# B&R Automation Studio project RS15_RX_30005_r00 (part 5)

#### A5_AutomatCyclic.st - Cyclic code
```iecst
 (********************************************************************
 * COPYRIGHT -- Microsoft
 ********************************************************************
 * Program: A5_Automat
 * File: A5_AutomatCyclic.st
 * Author: pkiel
 * Created: July 13, 2011
 ********************************************************************
 * Implementation of program A5_Automat
 ********************************************************************)

PROGRAM _CYCLIC

  // Synchro ratio Master/Slave
     // Master = Virtuel
     gA[5].rRSynNum := gRecipeActive.Repeat ;
     gA[5].rRSynDen := g_rSizeEntryPullRol_mm / 25.4 ;

  // Signal synchro Holding axis
  MC_BR_AutControl_0.Signal2 := gA[3].Ind_bSynchroOK                       AND
                                (MC_BR_AutControl_0.ActualStateIndex = 10) ;
  MC_BR_AutControl_0.Signal3 := NOT(gA[3].Ind_bSynchroOK) ;

  // Gear ratio assignement
  IF gReg[5].Enable THEN
    rGearValue := gReg[5].SP_Repeat * gA[5].UnitsPerInch ;
  ELSE
    rGearValue := gA5_GearValue ;
  END_IF

(**** STRAIGHT GEARED CAM AUTOMAT WITH GEARING UPDATE AND NO ABSOLUTE PHASE SYNCHRONIZATION ***)

(* Set Up Master Position Parameter ID *)
  //Synch_Request := gA[5].Cmd_SynchronizedMotion ;
  Synch_Request := gA[5].Cmd_SynchronizedMotion AND NOT(MC_BR_AutControl_0.Stop) ;  // D.M. 26/01/2012 RS26 Pyrollpack_14661 added because after guard fault it happened that Stop=1 and Synch_Request=1 => MC_BR_AutControl_0 makes fault 29256
	IF (Synch_Request AND NOT ParID_Ready) THEN
		MC_BR_InitMasterParIDTransfer_0.Master:=gA[9].Ident;
	    MC_BR_InitMasterParIDTransfer_0.Slave:=gA[5].Ident;
	    MC_BR_InitMasterParIDTransfer_0.MasterParID:=412;
	    MC_BR_InitMasterParIDTransfer_0.SlaveChannel:=0;
	    MC_BR_InitMasterParIDTransfer_0.Execute:=TRUE;
	    IF (MC_BR_InitMasterParIDTransfer_0.Done) THEN
	      MasterParID:=MC_BR_InitMasterParIDTransfer_0.ReceiveParID;
	      MC_BR_InitMasterParIDTransfer_0.Execute:=FALSE;
	      ParID_Ready:=1;
	    ELSIF (MC_BR_InitMasterParIDTransfer_0.Error) THEN
	    (*Store ErrorID in a variable,
	      ErrorID is reset on falling edge of 'Execute'*)
	      ErrorID:=MC_BR_InitMasterParIDTransfer_0.ErrorID;
	      ParID_Ready:=0;
	      MC_BR_InitMasterParIDTransfer_0.Execute:=FALSE;
	    END_IF
	END_IF
	MC_BR_InitMasterParIDTransfer_0();

(**** Initialize Automat Parameters Upon Automat Start Request ****)

	IF (EDGEPOS(ParID_Ready))THEN
		(*general automat parameter*)
			(*AutData.Master				:= gA[1].Ident;*)
			AutData.MasterParID			:= MasterParID;
			AutData.StartPosition		:= 0;
			AutData.StartInterval		:= gA[9].AxisPeriod;
			AutData.MaxMasterVelocity	:= gr_rMachMaxSpeed_BPM ;

		(*Automat STATE 0 Basis State*)
			AutData.State[0].Event[0].Type		  := ncST_END;
			AutData.State[0].Event[0].Attribute	:= ncAT_ONCE;
			//AutData.State[0].Event[0].NextState	:= 1;
      AutData.State[0].Event[0].NextState  := 10;

    //Waiting synchro Holding axis
      AutData.State[10].CamProfileIndex := 16#FFFF;
      AutData.State[10].MasterFactor    := REAL_TO_UDINT(gA[9].AxisPeriod);
      AutData.State[10].SlaveFactor     := 0;
      AutData.State[10].CompMode        := ncOFF;

      AutData.State[10].Event[0].Type      := ncSIGNAL3 ;
      AutData.State[10].Event[0].Attribute := ncAT_ONCE ;
      AutData.State[10].Event[0].NextState := 0;

      AutData.State[10].Event[0].Type      := ncSIGNAL2 ;
      AutData.State[10].Event[0].Attribute := ncAT_ONCE ;
      AutData.State[10].Event[0].NextState := 1;

		(*Automat STATE 1 Master/Slave Run*)
			AutData.State[1].CamProfileIndex := 16#FFFF;
			AutData.State[1].MasterFactor		 := REAL_TO_UDINT(gA[9].AxisPeriod);
			AutData.State[1].SlaveFactor		 := REAL_TO_UDINT(rGearValue);
			AutData.State[1].CompMode			   := ncOFF;

			AutData.State[1].Event[0].Type		:= ncST_END;
			AutData.State[1].Event[0].Attribute	:= ncST_END;
			AutData.State[1].Event[0].NextState	:= 1;

			AutData.State[1].Event[1].Type		:= ncST_END+ncNEGATIVE;
			AutData.State[1].Event[1].Attribute	:= ncST_END;
			AutData.State[1].Event[1].NextState	:= 1;

      AutData.State[1].Event[2].Type    := ncSIGNAL1;
      AutData.State[1].Event[2].Attribute  := ncAT_ONCE;
      AutData.State[1].Event[2].NextState  := 1;

      AutData.State[1].Event[3].Type    := ncSIGNAL3;
      AutData.State[1].Event[3].Attribute  := ncAT_ONCE;
      AutData.State[1].Event[3].NextState  := 0;

			MC_BR_AutControl_0.Enable 		:= 1;
			MC_BR_AutControl_0.AdrAutData 	:= ADR(AutData);
			MC_BR_AutControl_0.InitAutData 	:= 1;
	END_IF

		(* wait for initialization done *)
			IF ((MC_BR_AutControl_0.AutDataInitialized = 1)AND(Synch_Request)) THEN
				MC_BR_AutControl_0.InitAutData 	:= 0;
        uiMC_BR_AutControl_0_MemoErrorID := 0 ;
				AutomatStart := 1;
			END_IF
		(* check if error occured *)
			IF (MC_BR_AutControl_0.ErrorID <> 0) THEN
				MC_BR_AutControl_0.Enable := 0;
        uiMC_BR_AutControl_0_MemoErrorID := MC_BR_AutControl_0.ErrorID ;
			END_IF

(******************** ENABLE CAM-AUTOMAT **********************)
	IF (AutomatStart) THEN
			MC_BR_AutControl_0.Start := 1;
			AutomatStart := 0;
	END_IF

	IF (NOT Synch_Request) THEN
			MC_BR_AutControl_0.Stop := 1;
			MC_BR_AutControl_0.Start := 0;
			ParID_Ready := 0;
      IF (MC_BR_AutControl_0.Running=0) AND
         MC_BR_AutControl_0.Stop        THEN
        MC_BR_AutControl_0.Enable := 0;
        MC_BR_AutControl_0.Stop := 0;
      END_IF
   //*************************************************
   // D.M. 26/01/2012 RS26 Pyrollpack_14661 added because after guard fault it happened that Stop=1 and MC_BR_AutControl_0.Enable => not possible to finish MC_BR_AutControl_0 => program locked
      IF MC_BR_AutControl_0.Stop        AND
         NOT(MC_BR_AutControl_0.Enable) THEN
        MC_BR_AutControl_0.Enable := 1 ;
      END_IF
   //*************************************************
	END_IF
	gA[5].Ind_AutomatEnabled:=MC_BR_AutControl_0.Enable;
	gA[5].Ind_CurrentAutomatState:=MC_BR_AutControl_0.ActualStateIndex;
  gA[5].Ind_bSynchroOK := (MC_BR_AutControl_0.ActualStateIndex = 1) AND gA[5].Ind_SynchronizedMotion ;

(********************** MC_AUTCONTROL *************************)
	MC_BR_AutControl_0.Slave:= gA[5].Ident;
	MC_BR_AutControl_0();

(******************** UPDATE CAM-AUTOMAT STATE 1 **********************)
	MC_BR_InitAutState_0.MasterParID := MasterParID;
	MC_BR_InitAutState_0.Slave := gA[5].Ident;
	MC_BR_InitAutState_0.StateIndex := 1;
	MC_BR_InitAutState_0.CamProfileIndex := 16#FFFF;
	MC_BR_InitAutState_0.MasterFactor := REAL_TO_UDINT(gA[9].AxisPeriod);
	MC_BR_InitAutState_0.SlaveFactor := REAL_TO_DINT(rGearValue);
	MC_BR_InitAutState_0.CompMode := ncOFF;
	MC_BR_InitAutState_0.Execute := gA[5].Cmd_SynchronizedMotionUpdate;
	MC_BR_InitAutState_0();

  IF gA[5].Cmd_SynchronizedMotionUpdate THEN
    iTest_[2] := iTest_[2] + 1 ;
  END_IF

	IF (MC_BR_InitAutState_0.Done) THEN
		gA[5].Cmd_SynchronizedMotionUpdate:=0;
		MC_BR_AutControl_0.Signal1:=1;
    iTest_[0] := iTest_[0] + 1 ;
	ELSE
		MC_BR_AutControl_0.Signal1:=0;
	END_IF

  IF (MC_BR_InitAutState_0.Error) THEN
    gA[5].Cmd_SynchronizedMotionUpdate:=0;
    MC_BR_InitAutState_0.Execute := 0;
    iTest_[1] := iTest_[1] + 1 ;
  END_IF

END_PROGRAM
```

#### A5_Automat.var - Local variables
```iecst
(********************************************************************
 * COPYRIGHT -- Microsoft
 ********************************************************************
 * Program: A5_Automat
 * File: A5_Automat.var
 * Author: pkiel
 * Created: July 13, 2011
 ********************************************************************
 * Local variables of program A5_Automat
 ********************************************************************)
VAR
	AutData : MC_AUTDATA_TYP;
	AutomatStart : BOOL;
	ErrorID : UINT;
	MasterParID : UINT;
	MC_BR_AutControl_0 : MC_BR_AutControl;
  uiMC_BR_AutControl_0_MemoErrorID : UINT := 0 ;
	MC_BR_InitAutState_0 : MC_BR_InitAutState;
	MC_BR_InitMasterParIDTransfer_0 : MC_BR_InitMasterParIDTransfer;
	ParID_Ready : BOOL;
	Synch_Request : BOOL;

  iTest_ : ARRAY[0..9] OF INT ;
  rGearValue : REAL ;
END_VAR
```

### Program Logical/BagMachine_Section/EntryPull/Axis5/A5_Draw (IEC) - Axis Draw Calculations

#### A5_Draw.var - Local variables
```iecst
(********************************************************************
 * COPYRIGHT -- Microsoft
 ********************************************************************
 * Program: A5_Draw
 * File: A5_Draw.var
 * Author: pkiel
 * Created: July 13, 2011
 ********************************************************************
 * Local variables of program A5_Draw
 ********************************************************************)
VAR
	Draw_Old : REAL;
	First : BOOL;
  iLockEntryWebDraw : INT ;
  iBackColor : INT ;

  rEntry_Draw_Nul     : REAL := 0.0;
  rEntry_Draw_SP      : REAL := 0.0;
  HMI_rEntry_Draw_Set : REAL ;
END_VAR
```

### Program Logical/BagMachine_Section/EntryPull/Registration/A5_Reg1 (IEC) - Entry Pull Roll Registration

#### A5_Reg1Init.st
```iecst
(********************************************************************
 * COPYRIGHT -- Microsoft
 ********************************************************************
 * Program: A5_Reg1
 * File: A5_Reg1Init.st
 * Author: pkiel
 * Created: July 19, 2011
 ********************************************************************
 * Implementation of program A5_Reg1
 ********************************************************************)

PROGRAM _INIT

(*Set MC_BR_TouchProbe_0 Block to Capture Virtual Master Commanded Position (Par ID 412) *)
	TriggerRef_0.ProbeParID:=412;

(*Set MC_BR_TouchProbe_0 Block to Hardwired Trigger #1*)
	TriggerRef_0.EventSourceParID:=ACP10PAR_STAT_TRIGGER1;

(*Set MC_BR_TouchProbe_0 Block Trigger For Positive Edge *)
	TriggerRef_0.Edge:=0;

(*Set MC_BR_TouchProbe_1 Block to Capture Encoder #1 Actual Position (Par ID 91) *)
	TriggerRef_1.ProbeParID:=91;

(*Set MC_BR_TouchProbe_1 Block to Hardwired Trigger #1*)
	TriggerRef_1.EventSourceParID:=ACP10PAR_STAT_TRIGGER1;

(*Set MC_BR_TouchProbe_1 Block Trigger For Positive Edge *)
	TriggerRef_1.Edge:=0;

END_PROGRAM
```

### Program Logical/BagMachine_Section/EntryPull/Registration/A5_Reg2 (IEC) - Entry Pull Roll Registration Control

#### A5_Reg2.var
```iecst
(********************************************************************
 * COPYRIGHT -- Microsoft
 ********************************************************************
 * Program: A5_Reg2
 * File: A5_Reg2.var
 * Author: pkiel
 * Created: July 19, 2011
 ********************************************************************
 * Local variables of program A5_Reg2
 ********************************************************************)
VAR
	Background : UINT;
	Count : DINT;
	Diameter_Old : REAL;
	FirstAverage : BOOL;
	Foreground : UINT;
	Format_Old : REAL;
	HGW_Average_0 : HGW_Average;
	MissedMark_Count : DINT;
	Offset_Old : REAL;
	OutOfTolerance_Count : DINT;
	Repeat_Old : REAL;
END_VAR
```

### Package Logical/BagMachine_Section/ExitPull - Axis

### Program Logical/BagMachine_Section/ExitPull/Axis6/A6_Automat

#### A6_AutomatCyclic.st
```iecst
(********************************************************************
 * COPYRIGHT -- Microsoft
 ********************************************************************
 * Program: A6_Automat
 * File: A6_AutomatCyclic.st
 * Author: pkiel
 * Created: July 13, 2011
 ********************************************************************
 * Implementation of program A6_Automat
 ********************************************************************)

PROGRAM _CYCLIC

  // Synchro ratio Master/Slave
     // Master = EntryPull
     gA[6].rRSynNum := g_rSizeEntryPullRol_mm ;
     gA[6].rRSynDen := g_rSizeExitPullRol_mm ;

(**** STRAIGHT GEARED CAM AUTOMAT WITH GEARING UPDATE AND NO ABSOLUTE PHASE SYNCHRONIZATION ***)

(* Set Up Master Position Parameter ID *)
	Synch_Request := gA[6].Cmd_SynchronizedMotion;
  IF (Synch_Request AND NOT ParID_Ready) THEN
    MC_BR_InitMasterParIDTransfer_0.Master:=gA[5].Ident;
    MC_BR_InitMasterParIDTransfer_0.Slave:=gA[6].Ident;
    MC_BR_InitMasterParIDTransfer_0.MasterParID:=428;
    MC_BR_InitMasterParIDTransfer_0.SlaveChannel:=0;
	    MC_BR_InitMasterParIDTransfer_0.Execute:=TRUE;
	    IF (MC_BR_InitMasterParIDTransfer_0.Done) THEN
	      MasterParID:=MC_BR_InitMasterParIDTransfer_0.ReceiveParID;
	      MC_BR_InitMasterParIDTransfer_0.Execute:=FALSE;
	      ParID_Ready:=1;
	    ELSIF (MC_BR_InitMasterParIDTransfer_0.Error) THEN
	    (*Store ErrorID in a variable,
	      ErrorID is reset on falling edge of 'Execute'*)
	      ErrorID:=MC_BR_InitMasterParIDTransfer_0.ErrorID;
	      ParID_Ready:=0;
	      MC_BR_InitMasterParIDTransfer_0.Execute:=FALSE;
	    END_IF
	END_IF
	MC_BR_InitMasterParIDTransfer_0();

(**** Initialize Automat Parameters Upon Automat Start Request ****)

	IF (EDGEPOS(ParID_Ready))THEN
		(*general automat parameter*)
			(*AutData.Master				:= gA[1].Ident;*)
			AutData.MasterParID			:= MasterParID;
			AutData.StartPosition		:= 0;
			AutData.StartInterval		:= gA[5].AxisPeriod;
			AutData.MaxMasterVelocity	:= gr_rMachMaxSpeed_BPM ;

		(*Automat STATE 0 Basis State*)
			AutData.State[0].Event[0].Type		:= ncST_END;
			AutData.State[0].Event[0].Attribute	:= ncAT_ONCE;
			AutData.State[0].Event[0].NextState	:= 1;

		(*Automat STATE 1 Master/Slave Run*)
			AutData.State[1].CamProfileIndex	:= 16#FFFF;
      //AutData.State[1].MasterFactor    := REAL_TO_UDINT(gA[5].UnitsPerInch*rSizeEntryPullRol_In);
      AutData.State[1].MasterFactor    := REAL_TO_UDINT(gA[5].AxisPeriod);
			AutData.State[1].SlaveFactor		:= REAL_TO_UDINT(gA6_GearValue);
			AutData.State[1].CompMode			:= ncOFF;

			AutData.State[1].Event[0].Type		:= ncST_END;
			AutData.State[1].Event[0].Attribute	:= ncST_END;
			AutData.State[1].Event[0].NextState	:= 1;

			AutData.State[1].Event[1].Type		:= ncST_END+ncNEGATIVE;
			AutData.State[1].Event[1].Attribute	:= ncST_END;
			AutData.State[1].Event[1].NextState	:= 1;

			AutData.State[1].Event[2].Type		:= ncSIGNAL1;
			AutData.State[1].Event[2].Attribute	:= ncAT_ONCE;
			AutData.State[1].Event[2].NextState	:= 1;

			MC_BR_AutControl_0.Enable 		:= 1;
			MC_BR_AutControl_0.AdrAutData 	:= ADR(AutData);
			MC_BR_AutControl_0.InitAutData 	:= 1;
	END_IF

		(* wait for initialization done *)
			IF ((MC_BR_AutControl_0.AutDataInitialized = 1)AND(Synch_Request)) THEN
				MC_BR_AutControl_0.InitAutData 	:= 0;
				AutomatStart := 1;
			END_IF
		(* check if error occured *)
			IF (MC_BR_AutControl_0.ErrorID <> 0) THEN
				MC_BR_AutControl_0.Enable := 0;
			END_IF

(******************** ENABLE CAM-AUTOMAT **********************)
	IF (AutomatStart) THEN
			MC_BR_AutControl_0.Start := 1;
			AutomatStart := 0;
	END_IF

	IF (NOT Synch_Request) THEN
			MC_BR_AutControl_0.Stop := 1;
			MC_BR_AutControl_0.Start := 0;
			ParID_Ready := 0;
			IF (MC_BR_AutControl_0.Running=0) THEN
				MC_BR_AutControl_0.Enable := 0;
				MC_BR_AutControl_0.Stop := 0;
			END_IF
	END_IF
	gA[6].Ind_AutomatEnabled:=MC_BR_AutControl_0.Enable;
	gA[6].Ind_CurrentAutomatState:=MC_BR_AutControl_0.ActualStateIndex;
  gA[6].Ind_bSynchroOK := (MC_BR_AutControl_0.ActualStateIndex = 1) AND gA[6].Ind_SynchronizedMotion ;

(********************** MC_AUTCONTROL *************************)
	MC_BR_AutControl_0.Slave:= gA[6].Ident;
	MC_BR_AutControl_0();

(******************** UPDATE CAM-AUTOMAT STATE 1 **********************)
	MC_BR_InitAutState_0.MasterParID := MasterParID;
	MC_BR_InitAutState_0.Slave := gA[6].Ident;
	MC_BR_InitAutState_0.StateIndex := 1;
	MC_BR_InitAutState_0.CamProfileIndex := 16#FFFF;
  //MC_BR_InitAutState_0.MasterFactor := REAL_TO_UDINT(gA[5].UnitsPerInch*gRecipeActive.Repeat);
  MC_BR_InitAutState_0.MasterFactor := REAL_TO_UDINT(gA[5].AxisPeriod);
	MC_BR_InitAutState_0.SlaveFactor := REAL_TO_DINT(gA6_GearValue);
	MC_BR_InitAutState_0.CompMode := ncOFF;
	MC_BR_InitAutState_0.Execute := gA[6].Cmd_SynchronizedMotionUpdate;
	MC_BR_InitAutState_0();

	IF (MC_BR_InitAutState_0.Done) THEN
		gA[6].Cmd_SynchronizedMotionUpdate:=0;
		MC_BR_AutControl_0.Signal1:=1;
	ELSE
		MC_BR_AutControl_0.Signal1:=0;
	END_IF

	IF (MC_BR_InitAutState_0.Error) THEN
		gA[6].Cmd_SynchronizedMotionUpdate:=0;
		MC_BR_InitAutState_0.Execute := 0;
	END_IF

END_PROGRAM
```

### Program Logical/BagMachine_Section/ExitPull/Axis6/A6_Basic (IEC)

#### A6_BasicCyclic.st - Cyclic code
```iecst
(********************************************************************
 * COPYRIGHT -- Microsoft
 ********************************************************************
 * Program: A6_Basic
 * File: A6_BasicCyclic.st
 * Author: pkiel
 * Created: July 13, 2011
 ********************************************************************
 * Implementation of program A6_Basic
 ********************************************************************)

PROGRAM _CYCLIC

	IF (gA[6].Ident<>0) THEN

	(************************ READ DRIVE STATUS *************************)
	(* Access to the following bools:
	gA[x]_DriveStatus.Simulation			: If TRUE, simulation mode is active
	gA[x]_DriveStatus.NetworkInit			: If TRUE, the network is initialized
	gA[x]_DriveStatus.HomeSwitch			: If TRUE, the digital reference switch input is active
	gA[x]_DriveStatus.PosHWSwitch			: If TRUE, the positive hardware end switch is active
	gA[x]_DriveStatus.NegHWSwitch			: If TRUE, the negative hardware end switch is active
	gA[x]_DriveStatus.Trigger1				: If TRUE, the first trigger input is active
	gA[x]_DriveStatus.Trigger2				: If TRUE, the second trigger input is active
	gA[x]_DriveStatus.DriveEnable			: If TRUE, the enable input is active
	gA[x]_DriveStatus.ControllerReady		: If TRUE, the controller is ready to beturned on
	gA[x]_DriveStatus.ControllerStatus		: If TRUE, the controller is turned on (Same as MC_Power.Status)
	gA[x]_DriveStatus.AxisError				: If TRUE, at least one error has occurred (not acknowledged)
	gA[x]_DriveStatus.LagWarning			: If TRUE, the lag error has exceeded the limit value specified for a warning*)
		MC_BR_ReadDriveStatus_0.Enable := 1;
		MC_BR_ReadDriveStatus_0.Axis := gA[6].Ident;
		MC_BR_ReadDriveStatus_0.AdrDriveStatus := ADR (DriveStatus);
		MC_BR_ReadDriveStatus_0();
		gA[6].Ind_Simulation		:=	DriveStatus.Simulation;
		gA[6].Ind_NetworkInit		:=	DriveStatus.NetworkInit;
		gA[6].Input_Home			:=	DriveStatus.HomeSwitch;
		gA[6].Input_PosHW			:=	DriveStatus.PosHWSwitch;
		gA[6].Input_NegHW			:=	DriveStatus.NegHWSwitch;
		gA[6].Input_Trigger1		:=	DriveStatus.Trigger1;
		gA[6].Input_Trigger2		:=	DriveStatus.Trigger2;
		gA[6].Input_DriveEnable		:=	DriveStatus.DriveEnable;
		gA[6].Ind_ControllerReady	:=	DriveStatus.ControllerReady;
		gA[6].Ind_ControllerStatus	:=	DriveStatus.ControllerStatus;
		gA[6].Error					:=	DriveStatus.AxisError;
		gA[6].Ind_LagWarning		:=	DriveStatus.LagWarning;

	(************************ READ AXIS ERROR **********************)
		MC_ReadAxisError_0.Enable := gA[6].Ind_NetworkInit;
		MC_ReadAxisError_0.Axis := gA[6].Ident;
		MC_ReadAxisError_0.DataAddress := ADR(gA[6].ErrorText);
		MC_ReadAxisError_0.DataLength := SIZEOF(gA[6].ErrorText);
		MC_ReadAxisError_0.DataObjectName := 'Error_Eng';
		MC_ReadAxisError_0();
		IF(MC_ReadAxisError_0.Valid) THEN
			gA[6].ErrorID := MC_ReadAxisError_0.AxisErrorID;
			gA[6].ErrorCount := MC_ReadAxisError_0.AxisErrorCount;
		END_IF
	(* Auto Acknowledge Errors *)
		IF (gA[6].Cmd_Reset AND (gA[6].ErrorCount<>0) AND NOT AutoAck) THEN
			AutoAck:=1;
		ELSE
			AutoAck:=0;
		END_IF
	(*Axis Error Acknowledge*)
		IF (EDGEPOS(AutoAck) OR EDGEPOS(gA[6].ErrorAck)) THEN
			MC_ReadAxisError_0.Acknowledge := 1;
		ELSE;
			MC_ReadAxisError_0.Acknowledge :=0;
		END_IF

	(************************ RESET AXIS ERROR **********************)
		IF (gA[6].Cmd_Reset AND (gA[6].ErrorCount=0) AND gA[6].ErrorStop) THEN
			MC_Reset_0.Execute:=1;
		END_IF
		IF (MC_Reset_0.Done) THEN
			MC_Reset_0.Execute:=0;
			gA[6].Cmd_Reset:=0;
			ResetError := 0;
		END_IF
		IF (MC_Reset_0.Error) THEN
			MC_Reset_0.Execute:=0;
			gA[6].Cmd_Reset:=0;
			ResetError := 1;
		END_IF
		MC_Reset_0.Axis:=gA[6].Ident;
		MC_Reset_0();

	(************************ READ AXIS STATUS *************************)
		MC_ReadStatus_0.Enable := gA[6].Ind_NetworkInit;
		MC_ReadStatus_0.Axis := gA[6].Ident;
		MC_ReadStatus_0();
		IF(MC_ReadStatus_0.Valid = TRUE)THEN
			gA[6].Ind_Enabled 			:= NOT (MC_ReadStatus_0.Disabled);
			gA[6].Ind_StandStill		:= MC_ReadStatus_0.StandStill;
			gA[6].Ind_Stopping			:= MC_ReadStatus_0.Stopping;
			gA[6].Ind_DiscreteMotion	:= MC_ReadStatus_0.DiscreteMotion;
			gA[6].Ind_ContinuousMotion	:= MC_ReadStatus_0.ContinuousMotion;
			gA[6].Ind_SynchronizedMotion:= MC_ReadStatus_0.SynchronizedMotion;
			gA[6].ErrorStop				:= MC_ReadStatus_0.Errorstop;
		END_IF

	(******************** INIT POSITION MODULUS  *********************)
		MC_BR_InitModPos_0.Execute:= InitModPosition;
		MC_BR_InitModPos_0.Axis:= gA[6].Ident;
		MC_BR_InitModPos_0.Period:= REAL_TO_UDINT(gA[6].AxisPeriod);
		MC_BR_InitModPos_0.Factor:=1;
		InitModPos_Done:=MC_BR_InitModPos_0.Done;
		MC_BR_InitModPos_0();

	(******************** INIT ENDLESS POSITION *********************)
		MC_BR_InitEndlessPosition_0.Execute:= InitModPos_Done;
		MC_BR_InitEndlessPosition_0.Axis:= gA[6].Ident;
		MC_BR_InitEndlessPosition_0.DataAddress:= ADR(gEndPosData[6]);
		IF (MC_BR_InitEndlessPosition_0.Done) THEN
			InitModPosition:=0;
			InitEndlessPosition:=0;
			HomeRestore:=1;
		END_IF
		MC_BR_InitEndlessPosition_0();

	(************************ HOME AXIS FIRST POWER UP **********************)
		IF (HomeRestore AND NOT gA6_FirstHomed) THEN
			MC_Home_0.Execute:=1;
		END_IF
		MC_Home_0.Axis:=gA[6].Ident;
		MC_Home_0.Position:=0;
		MC_Home_0.HomingMode:=mcHOME_DIRECT;
		IF (MC_Home_0.Done) THEN
			MC_Home_0.Execute:=0;
			gA6_FirstHomed:=1;
		END_IF
		MC_Home_0();

	(************************ HOME AXIS **********************)
		IF (gA6_FirstHomed) THEN
			MC_Home_1.Execute:=HomeRestore;
		END_IF
		MC_Home_1.Axis:=gA[6].Ident;
		MC_Home_1.Position:=0;
		MC_Home_1.HomingMode:=mcHOME_RESTORE_POS;
		IF (MC_Home_1.Done) THEN
			gA[6].Ind_Homed:=1;
			HomeRestore:=0;
		END_IF
		MC_Home_1();

	(******************** READ ACTUAL POSITION *********************)
		MC_ReadActualPosition_0.Enable:= gA[6].Ind_NetworkInit;
		MC_ReadActualPosition_0.Axis:= gA[6].Ident;
		MC_ReadActualPosition_0();
		IF(MC_ReadActualPosition_0.Valid = TRUE)THEN
			gA[6].PositionCount := MC_ReadActualPosition_0.Position;
			gA[6].PositionInch := gA[6].PositionCount/gA[6].UnitsPerInch;
			gA[6].PositionDeg := gA[6].PositionCount/gA[6].UnitsPerDeg;
		END_IF

	(******************** READ ACTUAL VELOCITY *********************)
		IF(MC_ReadActualVelocity_0.Error=TRUE) THEN
			MC_ReadActualVelocity_0.Enable:= 0;
		ELSE
			MC_ReadActualVelocity_0.Enable:= 1;
		END_IF
		MC_ReadActualVelocity_0.Axis:= gA[6].Ident;
		MC_ReadActualVelocity_0();
		IF(MC_ReadActualVelocity_0.Valid = TRUE)THEN
			//gA[6].ActualVelocity := MC_ReadActualVelocity_0.Velocity*60/gA[6].SP_MotorPPR;
      gA[6].ActualVelocity := MC_ReadActualVelocity_0.Velocity*60/gA[6].AxisPeriod ; // D.M. 03/08/2011 BrownPaper_14542  Need speed of the axis and not of the shaft of the motor
      IF ABS(gA[6].ActualVelocity>1) THEN // D.M. 03/08/2011 BrownPaper_14542 Add ABS because in case negative velocity Ind_InMotion = 0 instead of 1
				gA[6].Ind_InMotion:=1;
			ELSE
				gA[6].Ind_InMotion:=0;
			END_IF
		END_IF

	(******************** READ ACTUAL TORQUE *********************)
		IF(MC_ReadActualTorque_0.Error=TRUE) THEN
			MC_ReadActualTorque_0.Enable:= 0;
		ELSE
			MC_ReadActualTorque_0.Enable:= 1;
		END_IF
		MC_ReadActualTorque_0.Axis:= gA[6].Ident;
		MC_ReadActualTorque_0();
		IF(MC_ReadActualTorque_0.Valid = TRUE)THEN
			gA[6].ActualTorque := MC_ReadActualTorque_0.Torque;
		END_IF

	(************************ ENABLE AXIS **********************)
		MC_Power_0.Axis:=gA[6].Ident;
		IF (MC_Power_0.Error=0) THEN
			MC_Power_0.Enable:=gA[6].Cmd_Enable;
		ELSE;
			MC_Power_0.Enable:=0;
		END_IF;
		MC_Power_0();

	(************************ AXIS VELOCITY MOVE **********************)
		MC_MoveVelocity_0.Axis:=gA[6].Ident;
		MC_MoveVelocity_0.Velocity:=gA[6].SP_Velocity*gA[6].AxisPeriod/60;
		MC_MoveVelocity_0.Acceleration:=gA[6].SP_Accel;
		MC_MoveVelocity_0.Deceleration:=gA[6].SP_Decel;
		MC_MoveVelocity_0.Direction:=mcPOSITIVE_DIR;
		IF ((EDGEPOS(gA[6].Cmd_ContinuousMotion)) OR (EDGEPOS(gA[6].Cmd_ContinuousMotionUpdate))) THEN
			MC_MoveVelocity_0.Execute:=1;
		ELSE
			MC_MoveVelocity_0.Execute:=0;
		END_IF;
		MC_MoveVelocity_0();

  //************************ AXIS OVERRIDE **********************
    MC_SetOverride_0.Axis      := gA[6].Ident ;
    MC_SetOverride_0.Enable    := gA[6].Cmd_Override ;
    MC_SetOverride_0.VelFactor := gA[6].rSP_OverrideV ;
    MC_SetOverride_0.AccFactor := gA[6].rSP_OverrideA ;
    IF (MC_SetOverride_0.Enabled) OR
       (MC_SetOverride_0.Error)   THEN
      gA[6].Cmd_Override := 0 ;
    END_IF
    MC_SetOverride_0();

	(************************ AXIS STOP **********************)
		MC_Stop_0.Axis:=gA[6].Ident;
		IF (gA[6].Ind_ContinuousMotion AND (NOT gA[6].Cmd_ContinuousMotion) AND gAlarmsOK) THEN
			MC_Stop_0.Deceleration:=gA[6].SP_Decel;
			MC_Stop_0.Execute:=1;
		END_IF;
		IF (MC_Stop_0.Done OR MC_Stop_0.CommandAborted OR MC_Stop_0.Error) THEN
			MC_Stop_0.Execute:=0;
		END_IF;
		MC_Stop_0();

  (************************  ESTOP **********************)
    MC_Stop_1.Axis:=gA[6].Ident;
    IF EDGEPOS(g_bIndEStopStandstill) THEN
      MC_Stop_1.Deceleration:=gA[6].SP_EStopDecel;
      MC_Stop_1.Execute:=1;
    END_IF;
    IF (MC_Stop_1.Done OR MC_Stop_1.CommandAborted OR MC_Stop_1.Error) THEN
      MC_Stop_1.Execute:=0;
      gA[6].Cmd_EStopDisable := 1 ;
    END_IF;
    IF NOT(g_bIndEStopStandstill) THEN
      gA[6].Cmd_EStopDisable := 0 ;
    END_IF;
    MC_Stop_1();

		(************************ AXIS PHASE CONTROL (Inches) **********************)
		MC_BR_Phasing_0.Slave:=gA[6].Ident;
		IF (gA[6].Ind_SynchronizedMotion) THEN
			MC_BR_Phasing_0.Enable:=1;
		ELSE;
			MC_BR_Phasing_0.Enable:=0;
		END_IF;
		IF (gA[6].Cmd_PhaseOffset) THEN
			MC_BR_Phasing_0.InitData:=1;
			gA[6].Cmd_PhaseOffset:=0;
		ELSE
			MC_BR_Phasing_0.InitData:=0;
		END_IF
		MC_BR_Phasing_0.ApplicationMode:=mcMASTER_DISTANCE_BASED;
		MC_BR_Phasing_0.Shift:=gA[6].SP_PhaseOffset*gA[9].UnitsPerInch;
		MC_BR_Phasing_0.Velocity:=6*gA[6].AxisPeriod/60;
		MC_BR_Phasing_0.Acceleration:=gA[6].SP_Decel;
		MC_BR_Phasing_0.ApplicationDistance:=2*gA[9].AxisPeriod;
		MC_BR_Phasing_0.ShiftMode:=mcRELATIVE;
		MC_BR_Phasing_0();

	END_IF

END_PROGRAM
```

#### A6_BasicInit.st - Initialization code
```iecst
(********************************************************************
 * COPYRIGHT -- Microsoft
 ********************************************************************
 * Program: A6_Basic
 * File: A6_BasicInit.st
 * Author: pkiel
 * Created: July 13, 2011
 ********************************************************************
 * Implementation of program A6_Basic
 ********************************************************************)

PROGRAM _INIT

	(* Axis Setpoint Variables *)
		gA[6].SP_MotorPPR := 18000;
		gA[6].SP_GearBoxInput:= 2;
		gA[6].SP_GearBoxOutput:= 1;
		gA[6].AxisPeriod := (gA[6].SP_MotorPPR*gA[6].SP_GearBoxInput/gA[6].SP_GearBoxOutput);
		gA[6].UnitsPerDeg := gA[6].AxisPeriod/360;
		gA[6].SP_Accel := 0.2*gA[6].AxisPeriod;
		gA[6].SP_Decel := 0.4*gA[6].AxisPeriod;
		gA[6].SP_EStopDecel := 1000.0*gA[6].AxisPeriod; // Stop axis from 1000 tr/min in 1s
		(* Theoretical Perimeter = 320mm *)
		gA[6].UnitsPerInch := (gA[6].AxisPeriod*25.4) / g_rSizeExitPullRol_mm ;
    gA[6].rSP_CorPosVel := 0.0 ;
    gA[6].rSP_OverrideV := 1.0 ;
    gA[6].rSP_OverrideA := 1.0 ;
    gA[6].Cmd_EStopDisable := 0 ;

	(* access master axis *)
		AxisErrorNcAccess := ncaccess(ncACP10MAN, ADR('Axis6'), ADR(gA[6].Ident));

	(* Trigger Initialization Of ModPosition *)
		InitModPosition:=1;

END_PROGRAM
```

### Program Logical/BagMachine_Section/ExitPull/Axis6/A6_Control (IEC)

#### A6_Control.var - Local variables
```iecst
(********************************************************************
 * COPYRIGHT -- Microsoft
 ********************************************************************
 * Program: A6_Control
 * File: A6_Control.var
 * Author: pkiel
 * Created: July 13, 2011
 ********************************************************************
 * Local variables of program A6_Control
 ********************************************************************)
VAR
	Synch_Permissive : BOOL;
	TOF_0 : TOF;
END_VAR
```

### Program Logical/BagMachine_Section/ExitPull/Axis6/A6_Draw (IEC)

#### A6_DrawCyclic.st - Cyclic code
```iecst
(********************************************************************
 * COPYRIGHT -- Microsoft
 ********************************************************************
 * Program: A6_Draw
 * File: A6_DrawCyclic.st
 * Author: pkiel
 * Created: July 13, 2011
 ********************************************************************
 * Implementation of program A6_Draw
 ********************************************************************)

PROGRAM _CYCLIC

  // Draw Setpoint Limits *)
	gRecipeActive.Exit_Draw := LIMIT(-100,gRecipeActive.Exit_Draw,100);

(* Manual Draw Calculations *)
	IF (((gRecipeActive.Exit_Draw <> Draw_Old) OR (NOT First) OR gRepeatChange) AND gA[6].Ind_SynchronizedMotion) THEN
   // gA6_GearValue := gA[6].UnitsPerInch * gRecipeActive.Repeat * (1.0+(gr_rMaxRangeWebDraw * 0.01 * gRecipeActive.Exit_Draw * 0.01));
    gA6_GearValue := gA[6].AxisPeriod * g_rSizeEntryPullRol_mm/g_rSizeExitPullRol_mm * (1.0+(gr_rMaxRangeWebDraw * 0.01 * gRecipeActive.Exit_Draw * 0.01));
    Draw_Old := gRecipeActive.Exit_Draw;
		First :=1;
		IF(gA[6].Ind_SynchronizedMotion) THEN
			gA[6].Cmd_SynchronizedMotionUpdate := 1;
		END_IF
	END_IF

END_PROGRAM
```

- Data object Logical/BagMachine_Section/ExitPull/Axis6/A6_Init (Ax) (no source held here)

### Data object Logical/BagMachine_Section/ExitPull/Axis6/A6_Par (Apt)

#### A6_Par.apt
```
AcoposParameterTable:
  Root Parameters:
    110 = ncSW_OFF (Name=CMD_SIMULATION)  // Simulation mode: Command
    128 = 1 (Name=SGEN_SW_END_IGNORE)  // SGEN_SW_END_IGNORE
```

### Program Logical/BagMachine_Section/ExitPull/ExitNip (IEC)

#### ExitNip.var - Local variables
```iecst
(********************************************************************
 * COPYRIGHT -- Microsoft
 ********************************************************************
 * Program: ExitNip
 * File: ExitNip.var
 * Author: pkiel
 * Created: July 20, 2011
 ********************************************************************
 * Local variables of program ExitNip
 ********************************************************************)

VAR
  bQ_SOL_WebExitNip : BOOL ;
END_VAR

VAR CONSTANT

END_VAR
```

### Package Logical/BagMachine_Section/Drum - Axis

### Program Logical/BagMachine_Section/Drum/Axis7/A7_Automat (IEC)

#### A7_Automat.var - Local variables
```iecst
(********************************************************************
 * COPYRIGHT -- Microsoft
 ********************************************************************
 * Program: A7_Automat
 * File: A7_Automat.var
 * Author: pkiel
 * Created: July 13, 2011
 ********************************************************************
 * Local variables of program A7_Automat
 ********************************************************************)
VAR
	AutData : MC_AUTDATA_TYP;
	AutomatStart : BOOL;
	ErrorID : UINT;
	MasterOffset : REAL;
  MasterParID : UINT;
  uiMasterParID1 : UINT;
	MC_BR_AutControl_0 : MC_BR_AutControl;
  uiMC_BR_AutControl_0_MemoErrorID : UINT ;
  MC_BR_InitMasterParIDTransfer_0 : MC_BR_InitMasterParIDTransfer;
  MC_BR_InitMasterParIDTransfer_1 : MC_BR_InitMasterParIDTransfer;
  ParID_Ready : BOOL;
  ParID_Ready1 : BOOL;
	PositionMOD : DINT;
	PositionOffset : DINT;
	SlaveStartOffset : REAL;
	Synch_Request : BOOL;
  uiSP_MasterParID : UINT;
  uiiSP_Master : UDINT;
  uiiSlaveFactor : UDINT;
  uiiMasterFactor : UDINT;
  uiiMaster : UDINT;
  usiMemoStat : USINT ;
  iiMasterFactor5 : DINT;
  iiSlaveFactor5  : DINT;
  bCmdSynchroOn : BOOL ;
  bCmdSynchroOff : BOOL ;
  rMaCompDist : REAL ;
  rSPMaPos    : REAL ;
  rOffsetDeg  : REAL ;
  rSlCompDist : REAL ;
  rTemp_      : ARRAY[0..9] OF REAL ;
  bTest_      : ARRAY[0..9] OF BOOL ;
  rRepeatMetric : REAL;
  rSlave_AxisPeriod : REAL ;
END_VAR
```

### Program Logical/BagMachine_Section/Drum/Axis7/A7_Basic

#### A7_BasicInit.st
```iecst
(********************************************************************
 * COPYRIGHT -- Microsoft
 ********************************************************************
 * Program: A7_Basic
 * File: A7_BasicInit.st
 * Author: pkiel
 * Created: July 13, 2011
 ********************************************************************
 * Implementation of program A7_Basic
 ********************************************************************)

PROGRAM _INIT

	(* Axis Setpoint Variables *)
		gA[7].SP_MotorPPR := 12000;
		gA[7].SP_GearBoxInput:= 3;  (* Note: Actual gear ratio = 12:1...However there are 4 stations/rev which yields an effective ratio of 3:1 *)
		gA[7].SP_GearBoxOutput:= 1;
		gA[7].AxisPeriod := (gA[7].SP_MotorPPR*gA[7].SP_GearBoxInput/gA[7].SP_GearBoxOutput);
		gA[7].UnitsPerDeg := gA[7].AxisPeriod/360;
		gA[7].SP_Accel := 0.2*gA[7].AxisPeriod;
		gA[7].SP_Decel := 0.4*gA[7].AxisPeriod;
		gA[7].SP_EStopDecel := 1000.0*gA[7].AxisPeriod; // Stop axis from 1000 tr/min in 1s
    gA[7].HomeVelocity := 6*gA[7].AxisPeriod/60;
    gA[7].rSP_CorPosVel := 0.0 ;
    gA[7].rSP_OverrideV := 1.0 ;
    gA[7].rSP_OverrideA := 1.0 ;
    gA[7].Cmd_EStopDisable := 0 ;

	(* access master axis *)
		AxisErrorNcAccess := ncaccess(ncACP10MAN, ADR('Axis7'), ADR(gA[7].Ident));

	(* Trigger Initialization Of ModPosition *)
		InitModPosition:=1;

    g_bIndPhasDrumInact := 1 ;

END_PROGRAM
```

### Program Logical/BagMachine_Section/Drum/Axis7/A7_Control (IEC)

#### A7_ControlCyclic.ld - Cyclic code
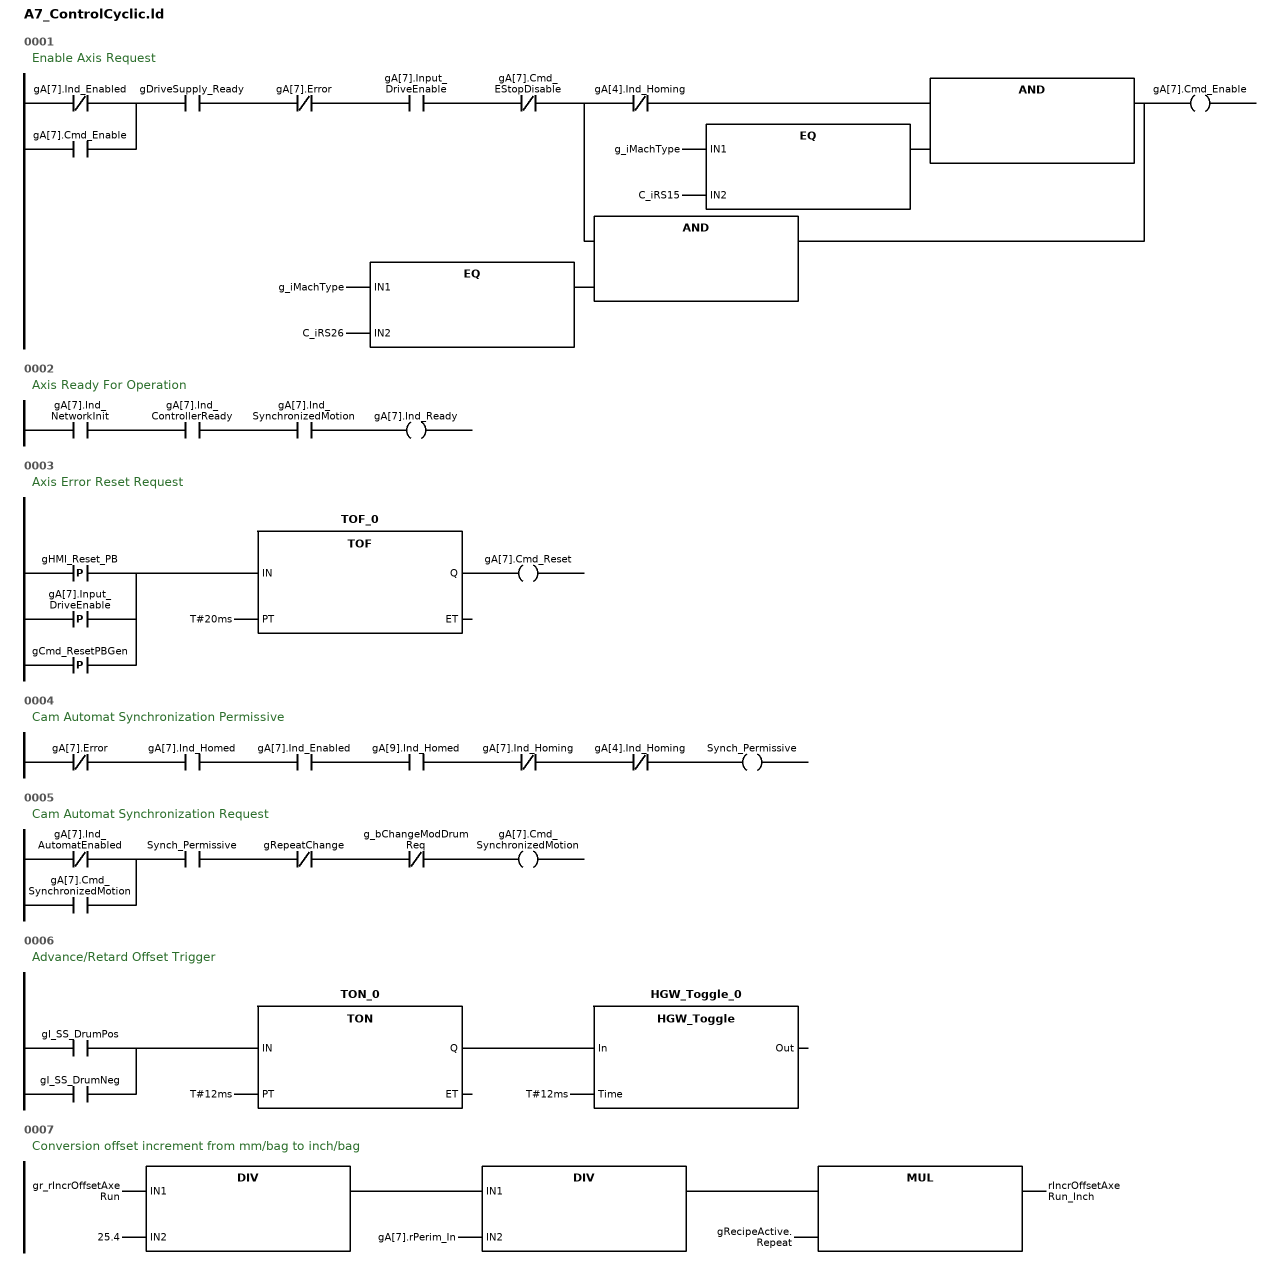
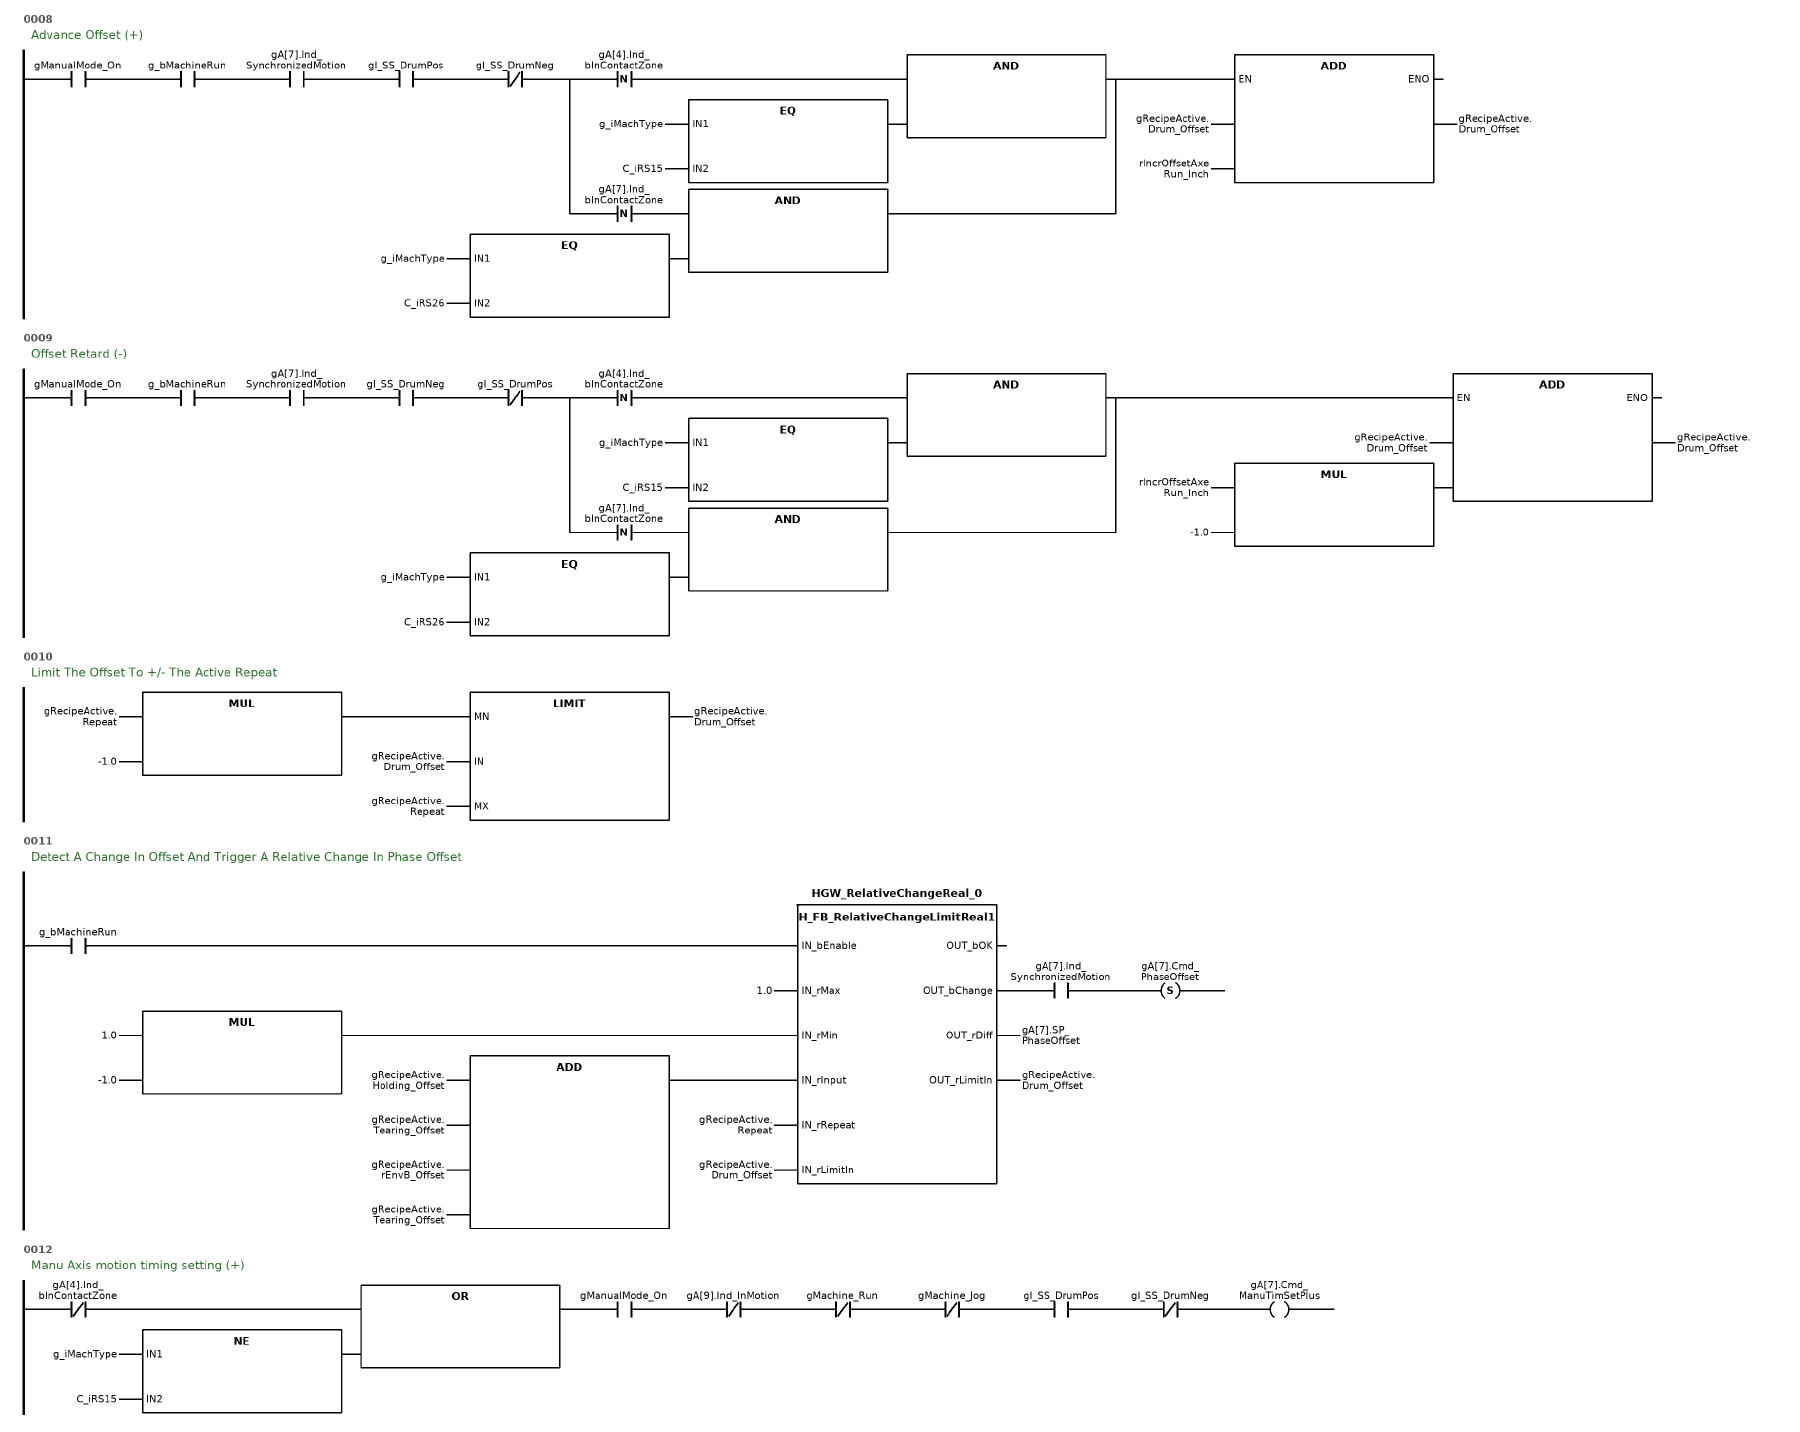
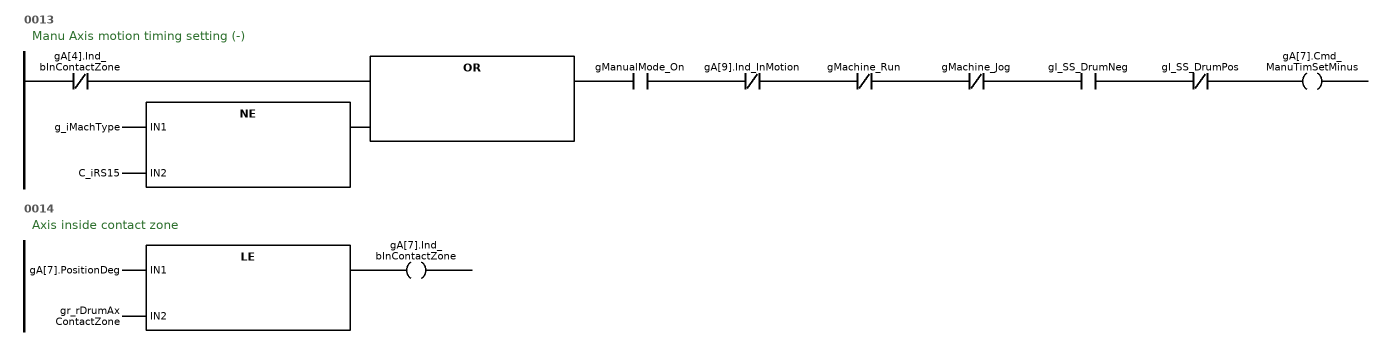
Ladder, written as Structured Text:
```iecst
(********************************************************************
 * COPYRIGHT -- Microsoft
 ********************************************************************
 * Program: A7_Control
 * File: A7_ControlCyclic.ld
 * Author: pkiel
 * Created: July 13, 2011
 ********************************************************************
 * Implementation of program A7_Control
 ********************************************************************)

PROGRAM _CYCLIC
VAR
    _p1 : BOOL;
    _e2 : R_TRIG;
    _e3 : R_TRIG;
    _e4 : R_TRIG;
    _p5 : BOOL;
    _e6 : F_TRIG;
    _e7 : F_TRIG;
    _p8 : BOOL;
    _e9 : F_TRIG;
    _e10 : F_TRIG;
END_VAR
(* Network 1: Enable Axis Request *)
_p1 := (NOT gA[7].Ind_Enabled OR gA[7].Cmd_Enable) AND gDriveSupply_Ready AND NOT gA[7].Error AND gA[7].Input_DriveEnable AND NOT gA[7].Cmd_EStopDisable;
gA[7].Cmd_Enable := _p1 AND ((NOT gA[4].Ind_Homing AND (g_iMachType = C_iRS15)) OR (g_iMachType = C_iRS26));

(* Network 2: Axis Ready For Operation *)
gA[7].Ind_Ready := gA[7].Ind_NetworkInit AND gA[7].Ind_ControllerReady AND gA[7].Ind_SynchronizedMotion;

(* Network 3: Axis Error Reset Request *)
_e2(CLK := gHMI_Reset_PB);
_e3(CLK := gA[7].Input_DriveEnable);
_e4(CLK := gCmd_ResetPBGen);
TOF_0(IN := _e2.Q OR _e3.Q OR _e4.Q, PT := T#20ms);
gA[7].Cmd_Reset := TOF_0.Q;

(* Network 4: Cam Automat Synchronization Permissive *)
Synch_Permissive := NOT gA[7].Error AND gA[7].Ind_Homed AND gA[7].Ind_Enabled AND gA[9].Ind_Homed AND NOT gA[7].Ind_Homing AND NOT gA[4].Ind_Homing;

(* Network 5: Cam Automat Synchronization Request *)
gA[7].Cmd_SynchronizedMotion := (NOT gA[7].Ind_AutomatEnabled OR gA[7].Cmd_SynchronizedMotion) AND Synch_Permissive AND NOT gRepeatChange AND NOT g_bChangeModDrumReq;

(* Network 6: Advance/Retard Offset Trigger *)
TON_0(IN := gI_SS_DrumPos OR gI_SS_DrumNeg, PT := T#12ms);
HGW_Toggle_0(In := TON_0.Q, Time := T#12ms);

(* Network 7: Conversion offset increment from mm/bag to inch/bag *)
rIncrOffsetAxeRun_Inch := ((gr_rIncrOffsetAxeRun / 25.4) / gA[7].rPerim_In) * gRecipeActive.Repeat;

(* Network 8: Advance Offset (+) *)
_p5 := gManualMode_On AND g_bMachineRun AND gA[7].Ind_SynchronizedMotion AND gI_SS_DrumPos AND NOT gI_SS_DrumNeg;
_e6(CLK := gA[4].Ind_bInContactZone);
_e7(CLK := gA[7].Ind_bInContactZone);
IF _p5 AND ((_e6.Q AND (g_iMachType = C_iRS15)) OR (_e7.Q AND (g_iMachType = C_iRS26))) THEN
    gRecipeActive.Drum_Offset := gRecipeActive.Drum_Offset + rIncrOffsetAxeRun_Inch;
END_IF;

(* Network 9: Offset Retard (-) *)
_p8 := gManualMode_On AND g_bMachineRun AND gA[7].Ind_SynchronizedMotion AND gI_SS_DrumNeg AND NOT gI_SS_DrumPos;
_e9(CLK := gA[4].Ind_bInContactZone);
_e10(CLK := gA[7].Ind_bInContactZone);
IF _p8 AND ((_e9.Q AND (g_iMachType = C_iRS15)) OR (_e10.Q AND (g_iMachType = C_iRS26))) THEN
    gRecipeActive.Drum_Offset := gRecipeActive.Drum_Offset + (rIncrOffsetAxeRun_Inch * -1.0);
END_IF;

(* Network 10: Limit The Offset To +/- The Active Repeat *)
gRecipeActive.Drum_Offset := LIMIT(MN := gRecipeActive.Repeat * -1.0, IN := gRecipeActive.Drum_Offset, MX := gRecipeActive.Repeat);

(* Network 11: Detect A Change In Offset And Trigger A Relative Change In Phase Offset *)
HGW_RelativeChangeReal_0(IN_bEnable := g_bMachineRun, IN_rMax := 1.0, IN_rMin := 1.0 * -1.0, IN_rInput := gRecipeActive.Holding_Offset + gRecipeActive.Tearing_Offset + gRecipeActive.rEnvB_Offset + gRecipeActive.Tearing_Offset, IN_rRepeat := gRecipeActive.Repeat, IN_rLimitIn := gRecipeActive.Drum_Offset);
IF HGW_RelativeChangeReal_0.OUT_bChange AND gA[7].Ind_SynchronizedMotion THEN
    gA[7].Cmd_PhaseOffset := TRUE;
END_IF;
gA[7].SP_PhaseOffset := HGW_RelativeChangeReal_0.OUT_rDiff;
gRecipeActive.Drum_Offset := HGW_RelativeChangeReal_0.OUT_rLimitIn;

(* Network 12: Manu Axis motion timing setting (+) *)
gA[7].Cmd_ManuTimSetPlus := (NOT gA[4].Ind_bInContactZone OR (g_iMachType <> C_iRS15)) AND gManualMode_On AND NOT gA[9].Ind_InMotion AND NOT gMachine_Run AND NOT gMachine_Jog AND gI_SS_DrumPos AND NOT gI_SS_DrumNeg;

(* Network 13: Manu Axis motion timing setting (-) *)
gA[7].Cmd_ManuTimSetMinus := (NOT gA[4].Ind_bInContactZone OR (g_iMachType <> C_iRS15)) AND gManualMode_On AND NOT gA[9].Ind_InMotion AND NOT gMachine_Run AND NOT gMachine_Jog AND gI_SS_DrumNeg AND NOT gI_SS_DrumPos;

(* Network 14: Axis inside contact zone *)
gA[7].Ind_bInContactZone := gA[7].PositionDeg <= gr_rDrumAxContactZone;
END_PROGRAM
```

### Program Logical/BagMachine_Section/Drum/Axis7/A7_Cycle (IEC)

#### A7_Cycle.var - Local variables
```iecst
(********************************************************************
 * COPYRIGHT -- .
 ********************************************************************
 * Program: A7_Cycle
 * File: A7_Cycle.var
 * Author: dominique
 * Created: August 01, 2011
 ********************************************************************
 * Local variables of program A7_Cycle
 ********************************************************************)

VAR
  bTest_          : ARRAY [0..9] OF BOOL ;
  iTest_          : ARRAY [0..9] OF INT ;
  rTempActPhasDeg : ARRAY[0..9] OF REAL ;
  rTempActOffsetInch : ARRAY[0..9] OF REAL ;
  rTemp_          : ARRAY[0..9] OF REAL ;
  stTON_01        : TON ;
END_VAR

VAR CONSTANT

END_VAR
```

### Data object Logical/BagMachine_Section/Drum/Axis7/A7_Par (Apt)

#### A7_Par.apt
```
AcoposParameterTable:
  Root Parameters:
    110 = ncSW_OFF (Name=CMD_SIMULATION)  // Simulation mode: Command
    128 = 1 (Name=SGEN_SW_END_IGNORE)  // SGEN_SW_END_IGNORE
    944 = 463 (Name=REFERENCE_SWITCH_PARID)  // REFERENCE_SWITCH_PARID
```

- Program Logical/BagMachine_Section/Drum/Axis7/A7_Ref (IEC) (no source held here)

### Package Logical/BagMachine_Section/ColdMicroPerf - Axis

### Program Logical/BagMachine_Section/ColdMicroPerf/CMPerf_Gen (IEC) - General Cold Micro Perf control

#### CMPerf_Gen.var
```iecst
(********************************************************************
 * COPYRIGHT -- .
 ********************************************************************
 * Program: CMPerf_Gen
 * File: CMPerf_en.var
 * Author: dominique
 * Created: November 05, 2011
 ********************************************************************
 * Local variables of program CMPerf_Gen
 ********************************************************************)

VAR CONSTANT

END_VAR

VAR
  HMI_CMPerf_bOnOffPB : BOOL ;

  bOnReq      : BOOL;
  bOffReq     : BOOL;
  bOn_PB      : BOOL ;
  bOff_PB     : BOOL ;

  bToolSizeLock : BOOL ;

END_VAR

VAR RETAIN
  HGW_2StatePB_0 : HGW_2StatePB;
END_VAR
```

#### CMPerf_GenInit.st
```iecst
(********************************************************************
 * COPYRIGHT -- .
 ********************************************************************
 * Program: CMPerf_Gen
 * File: CMPerf_GenInit.st
 * Author: dominique
 * Created: November 05, 2011
 ********************************************************************
 * Implementation of program CMPerf_Gen
 ********************************************************************)

PROGRAM _INIT

  // Cold Micro Perf On/Off
  HMI_CMPerf_bOnOffPB := gRecipeActive.bSelColdMicroPerfProd ;

  // Cold Micro Perf On/Off PB Colors
  HGW_2StatePB_0.BackColor_State0 := gYellow;
  HGW_2StatePB_0.ForeColor_State0 := gBlack;
  HGW_2StatePB_0.BackColor_State1 := gGreen;
  HGW_2StatePB_0.ForeColor_State1 := gBlack;

END_PROGRAM
```

### Data object Logical/BagMachine_Section/ColdMicroPerf/Axis8/A8_Init (Ax) - Servo Axis Initialization File

#### A8_Init.ax
```
InitParameter (Version=2.24.0, NcSwId=ACP10)
  ACP10AXIS_typ:
    dig_in:
      level:
        reference = ncACTIV_HI
        pos_hw_end = ncACTIV_HI
        neg_hw_end = ncACTIV_HI
        trigger1 = ncACTIV_HI
        trigger2 = ncACTIV_HI
    encoder_if:
      parameter:
        count_dir = ncINVERSE
        scaling:
          load:
            units = 12000
            rev_motor = 1
    limit:
      parameter:
        v_pos = 720000.0
        v_neg = 720000.0
        a1_pos = 5e+006
        a2_pos = 5e+006
        a1_neg = 5e+006
        a2_neg = 5e+006
        t_jolt = 0.0
        t_in_pos = 0.0
        pos_sw_end = 8388607
        neg_sw_end = -8388608
        ds_warning = 500.0
        ds_stop = 1000.0
        a_stop = 1e+030
        dv_stop = 0
        dv_stop_mode = ncOFF
    controller:
      mode = ncPOSITION
      position:
        kv = 300.0
        tn = 0.0
        t_predict = 0.0004
        t_total = 0.0012
        p_max = 1e+030
        i_max = 0.0
      speed:
        kv = 30.0
        tn = 0.0
        t_filter = 0.0
        isq_filter1:
          type = ncOFF
          a0 = 0.0
          a1 = 0.0
          b0 = 0.0
          b1 = 0.0
          b2 = 0.0
          c0_par_id = 0
          c1_par_id = 0
        isq_filter2:
          type = ncOFF
          a0 = 0.0
          a1 = 0.0
          b0 = 0.0
          b1 = 0.0
          b2 = 0.0
          c0_par_id = 0
          c1_par_id = 0
        isq_filter3:
          type = ncOFF
          a0 = 0.0
          a1 = 0.0
          b0 = 0.0
          b1 = 0.0
          b2 = 0.0
          c0_par_id = 0
          c1_par_id = 0
      uf:
        type = ncLINEAR
        auto_config = ncMOTOR_PAR
        u0 = 0.0
        un = 0.0
        fn = 50.0
        k_f_slip = 0.0
      ff:
        torque_load = 0.0
        torque_pos = 0.0
        torque_neg = 0.0
        kv_torque = 0.0
        inertia = 0.0
        t_filter_a = 0.0
    move:
      stop:
        parameter[0]:
          decel_ramp = ncA_LIMIT
          controller = ncON
        parameter[1]:
          decel_ramp = ncA_LIMIT
          controller = ncON
        parameter[2]:
          decel_ramp = ncA_LIMIT
          controller = ncON
        parameter[3]:
          decel_ramp = ncA_LIMIT
          controller = ncON
        quickstop:
          decel_ramp = ncA_LIMIT
        drive_error:
          decel_ramp = ncA_LIMIT
      homing:
        parameter:
          s = 0
          v_switch = 5000.0
          v_trigger = 500.0
          a = 50000.0
          mode = ncHOME_OFFSET
          edge_sw = ncPOSITIVE
          start_dir = ncPOSITIVE
          trigg_dir = ncPOSITIVE
          ref_pulse = ncOFF
          tr_s_block = 0.0
      basis:
        parameter:
          v_pos = 36000.0
          v_neg = 100000.0
          a1_pos = 50000.0
          a2_pos = 50000.0
          a1_neg = 50000.0
          a2_neg = 50000.0
    message:
      text:
        parameter:
          format = ncBREAK
          columns = 80
          data_modul = Error_Eng
```

### Data object Logical/BagMachine_Section/ColdMicroPerf/Axis8/A8_Par (Apt) - Servo Axis Parameter File

#### A8_Par.apt
```
AcoposParameterTable:
  Root Parameters:
    110 = ncSW_OFF (Name=CMD_SIMULATION)  // Simulation mode: Command
    128 = 1 (Name=SGEN_SW_END_IGNORE)  // SGEN_SW_END_IGNORE
    944 = 463 (Name=REFERENCE_SWITCH_PARID)  // Digital inputs: Parameter ID for reference switch
    390 = 565 (Name=UDC_NOMINAL, Unit=V)  // CTRL DC bus: Nominal voltage
```

### Program Logical/BagMachine_Section/ColdMicroPerf/Axis8/A8_Basic (IEC) - Basic Servo

#### A8_BasicCyclic.st
```iecst
(********************************************************************
 * COPYRIGHT -- Microsoft
 ********************************************************************
 * Program: A8_Basic
 * File: A8_BasicCyclic.st
 * Author: dominique
 * Created: November 03, 2011
 ********************************************************************
 * Implementation of program A8_Basic
 ********************************************************************)

PROGRAM _CYCLIC

	IF (gA[8].Ident<>0) THEN

	(************************ READ DRIVE STATUS *************************)
	(* Access to the following bools:
	gA[x]_DriveStatus.Simulation			: If TRUE, simulation mode is active
	gA[x]_DriveStatus.NetworkInit			: If TRUE, the network is initialized
	gA[x]_DriveStatus.HomeSwitch			: If TRUE, the digital reference switch input is active
	gA[x]_DriveStatus.PosHWSwitch			: If TRUE, the positive hardware end switch is active
	gA[x]_DriveStatus.NegHWSwitch			: If TRUE, the negative hardware end switch is active
	gA[x]_DriveStatus.Trigger1				: If TRUE, the first trigger input is active
	gA[x]_DriveStatus.Trigger2				: If TRUE, the second trigger input is active
	gA[x]_DriveStatus.DriveEnable			: If TRUE, the enable input is active
	gA[x]_DriveStatus.ControllerReady		: If TRUE, the controller is ready to beturned on
	gA[x]_DriveStatus.ControllerStatus		: If TRUE, the controller is turned on (Same as MC_Power.Status)
	gA[x]_DriveStatus.AxisError				: If TRUE, at least one error has occurred (not acknowledged)
	gA[x]_DriveStatus.LagWarning			: If TRUE, the lag error has exceeded the limit value specified for a warning*)
		MC_BR_ReadDriveStatus_0.Enable := 1;
		MC_BR_ReadDriveStatus_0.Axis := gA[8].Ident;
		MC_BR_ReadDriveStatus_0.AdrDriveStatus := ADR (DriveStatus);
		MC_BR_ReadDriveStatus_0();
		gA[8].Ind_Simulation		:=	DriveStatus.Simulation;
		gA[8].Ind_NetworkInit		:=	DriveStatus.NetworkInit;
		gA[8].Input_Home			:=	DriveStatus.HomeSwitch;
		gA[8].Input_PosHW			:=	DriveStatus.PosHWSwitch;
		gA[8].Input_NegHW			:=	DriveStatus.NegHWSwitch;
		gA[8].Input_Trigger1		:=	DriveStatus.Trigger1;
		gA[8].Input_Trigger2		:=	DriveStatus.Trigger2;
		gA[8].Input_DriveEnable		:=	DriveStatus.DriveEnable;
		gA[8].Ind_ControllerReady	:=	DriveStatus.ControllerReady;
		gA[8].Ind_ControllerStatus	:=	DriveStatus.ControllerStatus;
		gA[8].Error					:=	DriveStatus.AxisError;
		gA[8].Ind_LagWarning		:=	DriveStatus.LagWarning;

	(************************ READ AXIS ERROR **********************)
		MC_ReadAxisError_0.Enable := gA[8].Ind_NetworkInit;
		MC_ReadAxisError_0.Axis := gA[8].Ident;
		MC_ReadAxisError_0.DataAddress := ADR(gA[8].ErrorText);
		MC_ReadAxisError_0.DataLength := SIZEOF(gA[8].ErrorText);
		MC_ReadAxisError_0.DataObjectName := 'Error_Eng';
		MC_ReadAxisError_0();
		IF(MC_ReadAxisError_0.Valid) THEN
			gA[8].ErrorID := MC_ReadAxisError_0.AxisErrorID;
			gA[8].ErrorCount := MC_ReadAxisError_0.AxisErrorCount;
		END_IF
	(* Auto Acknowledge Errors *)
		IF (gA[8].Cmd_Reset AND (gA[8].ErrorCount<>0) AND NOT AutoAck) THEN
			AutoAck:=1;
		ELSE
			AutoAck:=0;
		END_IF
	(*Axis Error Acknowledge*)
		IF (EDGEPOS(AutoAck) OR EDGEPOS(gA[8].ErrorAck)) THEN
			MC_ReadAxisError_0.Acknowledge := 1;
		ELSE;
			MC_ReadAxisError_0.Acknowledge :=0;
		END_IF

	(************************ RESET AXIS ERROR **********************)
		IF (gA[8].Cmd_Reset AND (gA[8].ErrorCount=0) AND gA[8].ErrorStop) THEN
			MC_Reset_0.Execute:=1;
		END_IF
		IF (MC_Reset_0.Done) THEN
			MC_Reset_0.Execute:=0;
			gA[8].Cmd_Reset:=0;
			ResetError := 0;
		END_IF
		IF (MC_Reset_0.Error) THEN
			MC_Reset_0.Execute:=0;
			gA[8].Cmd_Reset:=0;
			ResetError := 1;
		END_IF
		MC_Reset_0.Axis:=gA[8].Ident;
		MC_Reset_0();

	(************************ READ AXIS STATUS *************************)
		MC_ReadStatus_0.Enable := gA[8].Ind_NetworkInit;
		MC_ReadStatus_0.Axis := gA[8].Ident;
		MC_ReadStatus_0();
		IF(MC_ReadStatus_0.Valid = TRUE)THEN
			gA[8].Ind_Enabled 			:= NOT (MC_ReadStatus_0.Disabled);
			gA[8].Ind_StandStill		:= MC_ReadStatus_0.StandStill;
			gA[8].Ind_Stopping			:= MC_ReadStatus_0.Stopping;
			gA[8].Ind_DiscreteMotion	:= MC_ReadStatus_0.DiscreteMotion;
			gA[8].Ind_ContinuousMotion	:= MC_ReadStatus_0.ContinuousMotion;
			gA[8].Ind_SynchronizedMotion:= MC_ReadStatus_0.SynchronizedMotion;
			gA[8].ErrorStop				:= MC_ReadStatus_0.Errorstop;
		END_IF

	(******************** INIT POSITION MODULUS  *********************)
		MC_BR_InitModPos_0.Execute:= InitModPosition;
		MC_BR_InitModPos_0.Axis:= gA[8].Ident;
		MC_BR_InitModPos_0.Period:= REAL_TO_UDINT(gA[8].AxisPeriod);
		MC_BR_InitModPos_0.Factor:=1;
		InitModPos_Done:=MC_BR_InitModPos_0.Done;
		MC_BR_InitModPos_0();

	(******************** INIT ENDLESS POSITION *********************)
		MC_BR_InitEndlessPosition_0.Execute:= InitModPos_Done;
		MC_BR_InitEndlessPosition_0.Axis:= gA[8].Ident;
		MC_BR_InitEndlessPosition_0.DataAddress:= ADR(gEndPosData[8]);
		IF (MC_BR_InitEndlessPosition_0.Done) THEN
			InitModPosition:=0;
			InitEndlessPosition:=0;
			HomeRestore:=1;
		END_IF
		MC_BR_InitEndlessPosition_0();

	(************************ HOME AXIS FIRST POWER UP **********************)
		IF (HomeRestore AND NOT gA8_FirstHomed) THEN
			MC_Home_0.Execute:=1;
		END_IF
		MC_Home_0.Axis:=gA[8].Ident;
		MC_Home_0.Position:=0;
		MC_Home_0.HomingMode:=mcHOME_DIRECT;
		IF (MC_Home_0.Done) THEN
			MC_Home_0.Execute:=0;
			gA8_FirstHomed:=1;
		END_IF
		MC_Home_0();

	(************************ HOME AXIS **********************)
		IF (gA8_FirstHomed) THEN
			MC_Home_1.Execute:=HomeRestore;
		END_IF
		MC_Home_1.Axis:=gA[8].Ident;
		MC_Home_1.Position:=0;
		MC_Home_1.HomingMode:=mcHOME_RESTORE_POS;
		IF (MC_Home_1.Done) THEN
			gA[8].Ind_Homed:=1;
			HomeRestore:=0;
		END_IF
		MC_Home_1();

	(******************** READ ACTUAL POSITION *********************)
		MC_ReadActualPosition_0.Enable:= gA[8].Ind_NetworkInit;
		MC_ReadActualPosition_0.Axis:= gA[8].Ident;
		MC_ReadActualPosition_0();
		IF(MC_ReadActualPosition_0.Valid = TRUE)THEN
			gA[8].PositionCount := MC_ReadActualPosition_0.Position;
			gA[8].PositionInch := gA[8].PositionCount/gA[8].UnitsPerInch;
			gA[8].PositionDeg := gA[8].PositionCount/gA[8].UnitsPerDeg;
		END_IF

	(******************** READ ACTUAL VELOCITY *********************)
		IF(MC_ReadActualVelocity_0.Error=TRUE) THEN
			MC_ReadActualVelocity_0.Enable:= 0;
		ELSE
			MC_ReadActualVelocity_0.Enable:= 1;
		END_IF
		MC_ReadActualVelocity_0.Axis:= gA[8].Ident;
		MC_ReadActualVelocity_0();
		IF(MC_ReadActualVelocity_0.Valid = TRUE)THEN
			//gA[8].ActualVelocity := MC_ReadActualVelocity_0.Velocity*60/gA[8].SP_MotorPPR;
      gA[8].ActualVelocity := MC_ReadActualVelocity_0.Velocity*60/gA[8].AxisPeriod ; // D.M. 03/08/2011 BrownPaper_14542  Need speed of the axis and not of the shaft of the motor
      IF ABS(gA[8].ActualVelocity>1) THEN // D.M. 03/08/2011 BrownPaper_14542 Add ABS because in case negative velocity Ind_InMotion = 0 instead of 1
				gA[8].Ind_InMotion:=1;
			ELSE
				gA[8].Ind_InMotion:=0;
			END_IF
		END_IF

	(******************** READ ACTUAL TORQUE *********************)
		IF(MC_ReadActualTorque_0.Error=TRUE) THEN
			MC_ReadActualTorque_0.Enable:= 0;
		ELSE
			MC_ReadActualTorque_0.Enable:= 1;
		END_IF
		MC_ReadActualTorque_0.Axis:= gA[8].Ident;
		MC_ReadActualTorque_0();
		IF(MC_ReadActualTorque_0.Valid = TRUE)THEN
			gA[8].ActualTorque := MC_ReadActualTorque_0.Torque;
		END_IF

	(************************ ENABLE AXIS **********************)
		MC_Power_0.Axis:=gA[8].Ident;
		IF (MC_Power_0.Error=0) THEN
			MC_Power_0.Enable:=gA[8].Cmd_Enable;
		ELSE;
			MC_Power_0.Enable:=0;
		END_IF;
		MC_Power_0();

	(************************ AXIS VELOCITY MOVE **********************)
		MC_MoveVelocity_0.Axis:=gA[8].Ident;
		MC_MoveVelocity_0.Velocity:=gA[8].SP_Velocity*gA[8].AxisPeriod/60;
		MC_MoveVelocity_0.Acceleration:=gA[8].SP_Accel;
		MC_MoveVelocity_0.Deceleration:=gA[8].SP_Decel;
		MC_MoveVelocity_0.Direction:=mcPOSITIVE_DIR;
		IF ((EDGEPOS(gA[8].Cmd_ContinuousMotion)) OR (EDGEPOS(gA[8].Cmd_ContinuousMotionUpdate))) THEN
			MC_MoveVelocity_0.Execute:=1;
		ELSE
			MC_MoveVelocity_0.Execute:=0;
		END_IF;
		MC_MoveVelocity_0();

  //************************ AXIS OVERRIDE **********************
    MC_SetOverride_0.Axis      := gA[8].Ident ;
    MC_SetOverride_0.Enable    := gA[8].Cmd_Override ;
    MC_SetOverride_0.VelFactor := gA[8].rSP_OverrideV ;
    MC_SetOverride_0.AccFactor := gA[8].rSP_OverrideA ;
    IF (MC_SetOverride_0.Enabled) OR
       (MC_SetOverride_0.Error)   THEN
      gA[8].Cmd_Override := 0 ;
    END_IF
    MC_SetOverride_0();

	(************************ AXIS STOP **********************)
		MC_Stop_0.Axis:=gA[8].Ident;
		IF (gA[8].Ind_ContinuousMotion AND (NOT gA[8].Cmd_ContinuousMotion) AND gAlarmsOK) THEN
			MC_Stop_0.Deceleration:=gA[8].SP_Decel;
			MC_Stop_0.Execute:=1;
		END_IF;
		IF (MC_Stop_0.Done OR MC_Stop_0.CommandAborted OR MC_Stop_0.Error) THEN
			MC_Stop_0.Execute:=0;
		END_IF;
		MC_Stop_0();

  (************************  ESTOP **********************)
    MC_Stop_1.Axis:=gA[8].Ident;
    IF EDGEPOS(g_bIndEStopStandstill) THEN
      MC_Stop_1.Deceleration:=gA[8].SP_EStopDecel;
      MC_Stop_1.Execute:=1;
    END_IF;
    IF (MC_Stop_1.Done OR MC_Stop_1.CommandAborted OR MC_Stop_1.Error) THEN
      MC_Stop_1.Execute:=0;
      gA[8].Cmd_EStopDisable := 1 ;
    END_IF;
    IF NOT(g_bIndEStopStandstill) THEN
      gA[8].Cmd_EStopDisable := 0 ;
    END_IF;
    MC_Stop_1();

		(************************ AXIS PHASE CONTROL (Inches) **********************)
		MC_BR_Phasing_0.Slave:=gA[8].Ident;
		IF (gA[8].Ind_SynchronizedMotion) THEN
			MC_BR_Phasing_0.Enable:=1;
		ELSE;
			MC_BR_Phasing_0.Enable:=0;
		END_IF;
		IF (gA[8].Cmd_PhaseOffset) THEN
			MC_BR_Phasing_0.InitData:=1;
			gA[8].Cmd_PhaseOffset:=0;
		ELSE
			MC_BR_Phasing_0.InitData:=0;
		END_IF
		MC_BR_Phasing_0.ApplicationMode:=mcMASTER_DISTANCE_BASED;
		MC_BR_Phasing_0.Shift:=gA[8].SP_PhaseOffset*gA[9].UnitsPerInch;
		MC_BR_Phasing_0.Velocity:=6*gA[8].AxisPeriod/60;
		MC_BR_Phasing_0.Acceleration:=gA[8].SP_Decel;
		MC_BR_Phasing_0.ApplicationDistance:=2*gA[9].AxisPeriod;
		MC_BR_Phasing_0.ShiftMode:=mcRELATIVE;
		MC_BR_Phasing_0();

	END_IF

END_PROGRAM
```

### Program Logical/BagMachine_Section/ColdMicroPerf/Axis8/A8_Control (IEC) - Servo Control

#### A8_ControlCyclic.ld - Cyclic code
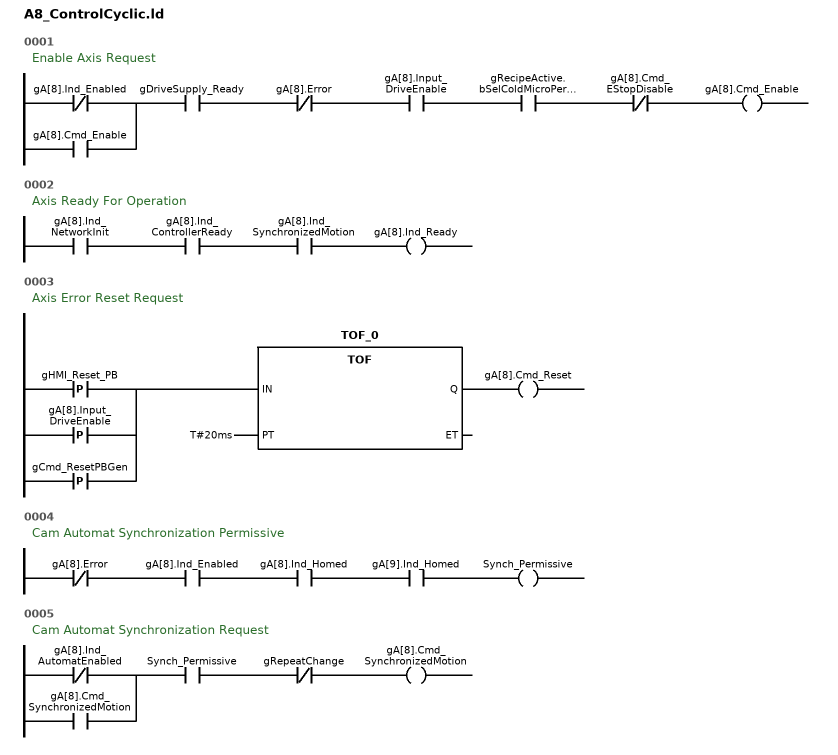
Ladder, written as Structured Text:
```iecst
(********************************************************************
 * COPYRIGHT -- Microsoft
 ********************************************************************
 * Program: A6_Control
 * File: A6_ControlCyclic.ld
 * Author: pkiel
 * Created: July 13, 2011
 ********************************************************************
 * Implementation of program A6_Control
 ********************************************************************)

PROGRAM _CYCLIC
VAR
    _e1 : R_TRIG;
    _e2 : R_TRIG;
    _e3 : R_TRIG;
END_VAR
(* Network 1: Enable Axis Request *)
gA[8].Cmd_Enable := (NOT gA[8].Ind_Enabled OR gA[8].Cmd_Enable) AND gDriveSupply_Ready AND NOT gA[8].Error AND gA[8].Input_DriveEnable AND gRecipeActive.bSelColdMicroPerfProd AND NOT gA[8].Cmd_EStopDisable;

(* Network 2: Axis Ready For Operation *)
gA[8].Ind_Ready := gA[8].Ind_NetworkInit AND gA[8].Ind_ControllerReady AND gA[8].Ind_SynchronizedMotion;

(* Network 3: Axis Error Reset Request *)
_e1(CLK := gHMI_Reset_PB);
_e2(CLK := gA[8].Input_DriveEnable);
_e3(CLK := gCmd_ResetPBGen);
TOF_0(IN := _e1.Q OR _e2.Q OR _e3.Q, PT := T#20ms);
gA[8].Cmd_Reset := TOF_0.Q;

(* Network 4: Cam Automat Synchronization Permissive *)
Synch_Permissive := NOT gA[8].Error AND gA[8].Ind_Enabled AND gA[8].Ind_Homed AND gA[9].Ind_Homed;

(* Network 5: Cam Automat Synchronization Request *)
gA[8].Cmd_SynchronizedMotion := (NOT gA[8].Ind_AutomatEnabled OR gA[8].Cmd_SynchronizedMotion) AND Synch_Permissive AND NOT gRepeatChange;
END_PROGRAM
```

### Program Logical/BagMachine_Section/ColdMicroPerf/Axis8/A8_Automat (IEC) - Cam Automat

#### A8_AutomatCyclic.st - Cyclic code
```iecst
(********************************************************************
 * COPYRIGHT -- Microsoft
 ********************************************************************
 * Program: A8_Automat
 * File: A8_AutomatCyclic.st
 * Author: dominique
 * Created: November 03, 2011
 ********************************************************************
 * Implementation of program A8_Automat
 ********************************************************************)

PROGRAM _CYCLIC

  // Synchro ratio Master/Slave
     // Master = EntryPull
     gA[8].rRSynNum := g_rSizeEntryPullRol_mm ;
     gA[8].rRSynDen := g_rSizeCMPerfRol_mm ;

  // Signal synchro Holding, Tearing and Drum axis
  MC_BR_AutControl_0.Signal1 := g_bIndSynchroHTD_OK ;

(**** STRAIGHT GEARED CAM AUTOMAT WITH GEARING UPDATE AND NO ABSOLUTE PHASE SYNCHRONIZATION ***)

(* Set Up Master Position Parameter ID *)
	Synch_Request := gA[8].Cmd_SynchronizedMotion;
	IF (Synch_Request AND NOT ParID_Ready) THEN
		MC_BR_InitMasterParIDTransfer_0.Master:=gA[5].Ident;
	    MC_BR_InitMasterParIDTransfer_0.Slave:=gA[8].Ident;
	    MC_BR_InitMasterParIDTransfer_0.MasterParID:=428;
	    MC_BR_InitMasterParIDTransfer_0.SlaveChannel:=0;
	    MC_BR_InitMasterParIDTransfer_0.Execute:=TRUE;
	    IF (MC_BR_InitMasterParIDTransfer_0.Done) THEN
	      MasterParID:=MC_BR_InitMasterParIDTransfer_0.ReceiveParID;
	      MC_BR_InitMasterParIDTransfer_0.Execute:=FALSE;
	      ParID_Ready:=1;
	    ELSIF (MC_BR_InitMasterParIDTransfer_0.Error) THEN
	    (*Store ErrorID in a variable,
	      ErrorID is reset on falling edge of 'Execute'*)
	      ErrorID:=MC_BR_InitMasterParIDTransfer_0.ErrorID;
	      ParID_Ready:=0;
	      MC_BR_InitMasterParIDTransfer_0.Execute:=FALSE;
	    END_IF
	END_IF
	MC_BR_InitMasterParIDTransfer_0();

(**** Initialize Automat Parameters Upon Automat Start Request ****)

	IF (EDGEPOS(ParID_Ready))THEN
		(*general automat parameter*)
			(*AutData.Master				:= gA[1].Ident;*)
			AutData.MasterParID			:= MasterParID;
			AutData.StartPosition		:= 0;
			AutData.StartInterval		:= gA[5].AxisPeriod;
			AutData.MaxMasterVelocity	:= gr_rMachMaxSpeed_BPM ;

		(*Automat STATE 0 Basis State*)
			AutData.State[0].Event[0].Type		:= ncST_END;
			AutData.State[0].Event[0].Attribute	:= ncAT_ONCE;
			AutData.State[0].Event[0].NextState	:= 1;

		(*Automat STATE 1 Master/Slave Run*)
			AutData.State[1].CamProfileIndex 	:= 16#FFFF;
      AutData.State[1].MasterFactor     := REAL_TO_UDINT(gA[5].AxisPeriod);
			AutData.State[1].SlaveFactor		  := REAL_TO_UDINT(gA8_GearValue);
			AutData.State[1].CompMode			    := ncOFF;

			AutData.State[1].Event[0].Type		:= ncST_END;
			AutData.State[1].Event[0].Attribute	:= ncST_END;
			AutData.State[1].Event[0].NextState	:= 1;

			AutData.State[1].Event[1].Type		:= ncST_END+ncNEGATIVE;
			AutData.State[1].Event[1].Attribute	:= ncST_END;
			AutData.State[1].Event[1].NextState	:= 1;

			AutData.State[1].Event[2].Type		:= ncSIGNAL1;
			AutData.State[1].Event[2].Attribute	:= ncAT_ONCE;
			AutData.State[1].Event[2].NextState	:= 1;

			MC_BR_AutControl_0.Enable 		:= 1;
			MC_BR_AutControl_0.AdrAutData 	:= ADR(AutData);
			MC_BR_AutControl_0.InitAutData 	:= 1;
	END_IF

		(* wait for initialization done *)
			IF ((MC_BR_AutControl_0.AutDataInitialized = 1)AND(Synch_Request)) THEN
				MC_BR_AutControl_0.InitAutData 	:= 0;
				AutomatStart := 1;
			END_IF
		(* check if error occured *)
			IF (MC_BR_AutControl_0.ErrorID <> 0) THEN
				MC_BR_AutControl_0.Enable := 0;
			END_IF

(******************** ENABLE CAM-AUTOMAT **********************)
	IF (AutomatStart) THEN
			MC_BR_AutControl_0.Start := 1;
			AutomatStart := 0;
	END_IF

	IF (NOT Synch_Request) THEN
			MC_BR_AutControl_0.Stop := 1;
			MC_BR_AutControl_0.Start := 0;
			ParID_Ready := 0;
			IF (MC_BR_AutControl_0.Running=0) THEN
				MC_BR_AutControl_0.Enable := 0;
				MC_BR_AutControl_0.Stop := 0;
			END_IF
	END_IF
	gA[8].Ind_AutomatEnabled:=MC_BR_AutControl_0.Enable;
	gA[8].Ind_CurrentAutomatState:=MC_BR_AutControl_0.ActualStateIndex;
  gA[8].Ind_bSynchroOK := (MC_BR_AutControl_0.ActualStateIndex = 1) AND gA[8].Ind_SynchronizedMotion ;

(********************** MC_AUTCONTROL *************************)
	MC_BR_AutControl_0.Slave:= gA[8].Ident;
	MC_BR_AutControl_0();

(******************** UPDATE CAM-AUTOMAT STATE 1 **********************)
	MC_BR_InitAutState_0.MasterParID := MasterParID;
	MC_BR_InitAutState_0.Slave := gA[8].Ident;
	MC_BR_InitAutState_0.StateIndex := 1;
	MC_BR_InitAutState_0.CamProfileIndex := 16#FFFF;
  MC_BR_InitAutState_0.MasterFactor := REAL_TO_UDINT(gA[5].AxisPeriod);
	MC_BR_InitAutState_0.SlaveFactor := REAL_TO_DINT(gA8_GearValue);
	MC_BR_InitAutState_0.CompMode := ncOFF;
	MC_BR_InitAutState_0.Execute := gA[8].Cmd_SynchronizedMotionUpdate;
	MC_BR_InitAutState_0();

	IF (MC_BR_InitAutState_0.Done) THEN
		gA[8].Cmd_SynchronizedMotionUpdate:=0;
		MC_BR_AutControl_0.Signal1:=1;
	ELSE
		MC_BR_AutControl_0.Signal1:=0;
	END_IF

	IF (MC_BR_InitAutState_0.Error) THEN
		gA[8].Cmd_SynchronizedMotionUpdate:=0;
		MC_BR_InitAutState_0.Execute := 0;
	END_IF

END_PROGRAM
```

### Program Logical/BagMachine_Section/ColdMicroPerf/Axis8/A8_Draw (IEC) - Axis Draw Calculations

#### A8_Draw.var - Local variables
```iecst
(********************************************************************
 * COPYRIGHT -- Microsoft
 ********************************************************************
 * Program: A8_Draw
 * File: A8_Draw.var
 * Author: dominique
 * Created: November 03, 2011
 ********************************************************************
 * Local variables of program A8_Draw
 ********************************************************************)
VAR
  Draw_Old : REAL;
	First : BOOL;

  rSizeTool_Old : REAL ;
END_VAR
```

### Package Logical/BagMachine_Section/EnvBag - Axis   Envelope Bag

### Program Logical/BagMachine_Section/EnvBag/EB_Gen (IEC) - General Envelope Bag control

#### EB_GenCyclic.st
```iecst
(********************************************************************
 * COPYRIGHT -- .
 ********************************************************************
 * Program: EB_Gen
 * File: EB_GenCyclic.st
 * Author: dominique
 * Created: November 21, 2011
 ********************************************************************
 * Implementation of program EB_Gen
 ********************************************************************)

PROGRAM _CYCLIC

  // ----------------------------------------------------------------------------------
  // On/Off Envelope Bag
  // Case On
  bEnvBOnReq := HMI_EnvB_bOnOffPB AND NOT(gRecipeActive.bSelEnvBProd) ;
  IF bEnvBOnReq THEN
    IF NOT(gA[9].Ind_InMotion) AND
       1                       THEN
      gRecipeActive.bSelEnvBProd := 1 ;
      HMI_EnvB_bWasteSucOnOffPB  := 1 ;
    ELSE
      gRecipeActive.bSelEnvBProd := 0 ;
      HMI_EnvB_bOnOffPB := 0 ;
    END_IF ;
  END_IF ;

  // Case Off
  bEnvBOffReq := NOT(HMI_EnvB_bOnOffPB) AND gRecipeActive.bSelEnvBProd ;
  IF bEnvBOffReq THEN
    IF NOT(gA[9].Ind_InMotion) AND
       1                       THEN
      gRecipeActive.bSelEnvBProd := 0 ;
      HMI_EnvB_bWasteSucOnOffPB  := 0 ;
    ELSE
      gRecipeActive.bSelEnvBProd := 1 ;
      HMI_EnvB_bOnOffPB := 1 ;
    END_IF ;
  END_IF ;

  // Indicator Envelope Bag selection change
  IF EDGE(gRecipeActive.bSelEnvBProd) THEN
    g_bEnvBagSelectChang := 1 ;
  END_IF ;

  // ----------------------------------------------------------------------------------
  // On/Off Waste Suction
  IF NOT(gRecipeActive.bSelEnvBProd) OR
     g_EnvB_bWasteSucMPAlarm         OR
     g_bIndEStop                     THEN
    HMI_EnvB_bWasteSucOnOffPB := 0 ;
  END_IF ;

  bWasteSucOn := HMI_EnvB_bWasteSucOnOffPB AND
                 gA[9].Ind_InMotion        AND
                 1                         ;

  stTOF_0(IN:=bWasteSucOn,PT:=T#60s) ;

  gQ_CR_EB_WasteSuction := stTOF_0.Q                 AND
                           HMI_EnvB_bWasteSucOnOffPB ;

  // ----------------------------------------------------------------------------------
  // Active indicator
  gA[12].bActive := gA[12].bInMach ;
  gA[13].bActive := gA[13].bInMach ;

END_PROGRAM
```

#### EB_GenInit.st
```iecst
(********************************************************************
 * COPYRIGHT -- .
 ********************************************************************
 * Program: FP_Gen
 * File: FP_GenInit.st
 * Author: dominique
 * Created: November 21, 2011
 ********************************************************************
 * Implementation of program FP_Gen
 ********************************************************************)

PROGRAM _INIT

  // Envelope Bag Off/On
  HMI_EnvB_bOnOffPB := gRecipeActive.bSelEnvBProd ;

END_PROGRAM
```

### Package Logical/BagMachine_Section/EnvBag/Axis12 - Envelope Bag Axis     EnvB  Axis

### Data object Logical/BagMachine_Section/EnvBag/Axis12/A12_Init (Ax) - Servo Axis Initialization File

#### A12_Init.ax
```
InitParameter (Version=2.24.0, NcSwId=ACP10)
  ACP10AXIS_typ:
    dig_in:
      level:
        reference = ncACTIV_HI
        pos_hw_end = ncACTIV_HI
        neg_hw_end = ncACTIV_HI
        trigger1 = ncACTIV_HI
        trigger2 = ncACTIV_HI
    encoder_if:
      parameter:
        count_dir = ncINVERSE
        scaling:
          load:
            units = 6000  // Units at the load     = 36000 / 6
            rev_motor = 1  // Motor revolutions    
    limit:
      parameter:
        v_pos = 600000.0
        v_neg = 600000.0
        a1_pos = 5e+006
        a2_pos = 5e+006
        a1_neg = 5e+006
        a2_neg = 5e+006
        t_jolt = 0.0
        t_in_pos = 0.0
        pos_sw_end = 8388607
        neg_sw_end = -8388608
        ds_warning = 500.0
        ds_stop = 1000.0
        a_stop = 1e+030
        dv_stop = 0
        dv_stop_mode = ncOFF
    controller:
      mode = ncPOSITION
      position:
        kv = 300.0
        tn = 0.0
        t_predict = 0.0004
        t_total = 0.0012
        p_max = 1e+030
        i_max = 0.0
      speed:
        kv = 30.0
        tn = 0.0
        t_filter = 0.0
        isq_filter1:
          type = ncOFF
          a0 = 0.0
          a1 = 0.0
          b0 = 0.0
          b1 = 0.0
          b2 = 0.0
          c0_par_id = 0
          c1_par_id = 0
        isq_filter2:
          type = ncOFF
          a0 = 0.0
          a1 = 0.0
          b0 = 0.0
          b1 = 0.0
          b2 = 0.0
          c0_par_id = 0
          c1_par_id = 0
        isq_filter3:
          type = ncOFF
          a0 = 0.0
          a1 = 0.0
          b0 = 0.0
          b1 = 0.0
          b2 = 0.0
          c0_par_id = 0
          c1_par_id = 0
      uf:
        type = ncLINEAR
        auto_config = ncMOTOR_PAR
        u0 = 0.0
        un = 0.0
        fn = 50.0
        k_f_slip = 0.0
      ff:
        torque_load = 0.0
        torque_pos = 0.0
        torque_neg = 0.0
        kv_torque = 0.0
        inertia = 0.0
        t_filter_a = 0.0
    move:
      stop:
        parameter[0]:
          decel_ramp = ncA_LIMIT
          controller = ncON
        parameter[1]:
          decel_ramp = ncA_LIMIT
          controller = ncON
        parameter[2]:
          decel_ramp = ncA_LIMIT
          controller = ncON
        parameter[3]:
          decel_ramp = ncA_LIMIT
          controller = ncON
        quickstop:
          decel_ramp = ncA_LIMIT
        drive_error:
          decel_ramp = ncA_LIMIT
      homing:
        parameter:
          s = 0
          v_switch = 7200.0
          v_trigger = 720.0
          a = 50000.0
          mode = ncHOME_OFFSET
          edge_sw = ncPOSITIVE
          start_dir = ncPOSITIVE
          trigg_dir = ncPOSITIVE
          ref_pulse = ncOFF
          tr_s_block = 0.0
      basis:
        parameter:
          v_pos = 36000.0
          v_neg = 100000.0
          a1_pos = 50000.0
          a2_pos = 50000.0
          a1_neg = 50000.0
          a2_neg = 50000.0
    message:
      text:
        parameter:
          format = ncBREAK
          columns = 80
          data_modul = Error_Eng
```

- Data object Logical/BagMachine_Section/EnvBag/Axis12/A12_Par (Apt) - Servo Axis Parameter File (no source held here)

### Program Logical/BagMachine_Section/EnvBag/Axis12/A12_Basic (IEC) - Basic Servo

#### A12_BasicCyclic.st - Cyclic code
```iecst
(********************************************************************
 * COPYRIGHT -- Microsoft
 ********************************************************************
 * Program: A12_Basic
 * File: A12_BasicCyclic.st
 * Author: dominique
 * Created: November 21, 2011
 ********************************************************************
 * Implementation of program A12_Basic
 ********************************************************************)

PROGRAM _CYCLIC

	gA[12].UnitsPerInch := gA[12].AxisPeriod/gRecipeActive.Repeat;
  gA[12].InchPerDeg := gA[12].UnitsPerDeg / gA[12].UnitsPerInch ;

  // Axis inside contact zone
  IF (gA[12].rRSynDen <> 0.0) THEN
    rA12PosTempAxis_deg := H_FC_Modulus (
                                IN_rMod := (360 * gA[12].rRSynNum/gA[12].rRSynDen) ,
                                IN_rVar := gA[12].PositionDeg
                                        ) ;
  END_IF
  IF (g_EnvB_iHoldTearEnvBCase<=3) THEN
    gA[12].Ind_bInContactZone := (rA12PosTempAxis_deg > 45.0)                        AND
                                 (rA12PosTempAxis_deg <= gr_rHoldAxContactZone+45.0) ;
  ELSE
    gA[12].Ind_bInContactZone := (rA12PosTempAxis_deg <= gr_rEnvBAxContactZone) ;
  END_IF

	IF (gA[12].Ident<>0) THEN

	(************************ READ DRIVE STATUS *************************)
	(* Access to the following bools:
	gA[x]_DriveStatus.Simulation			: If TRUE, simulation mode is active
	gA[x]_DriveStatus.NetworkInit			: If TRUE, the network is initialized
	gA[x]_DriveStatus.HomeSwitch			: If TRUE, the digital reference switch input is active
	gA[x]_DriveStatus.PosHWSwitch			: If TRUE, the positive hardware end switch is active
	gA[x]_DriveStatus.NegHWSwitch			: If TRUE, the negative hardware end switch is active
	gA[x]_DriveStatus.Trigger1				: If TRUE, the first trigger input is active
	gA[x]_DriveStatus.Trigger2				: If TRUE, the second trigger input is active
	gA[x]_DriveStatus.DriveEnable			: If TRUE, the enable input is active
	gA[x]_DriveStatus.ControllerReady		: If TRUE, the controller is ready to beturned on
	gA[x]_DriveStatus.ControllerStatus		: If TRUE, the controller is turned on (Same as MC_Power.Status)
	gA[x]_DriveStatus.AxisError				: If TRUE, at least one error has occurred (not acknowledged)
	gA[x]_DriveStatus.LagWarning			: If TRUE, the lag error has exceeded the limit value specified for a warning*)
		MC_BR_ReadDriveStatus_0.Enable := 1;
		MC_BR_ReadDriveStatus_0.Axis := gA[12].Ident;
		MC_BR_ReadDriveStatus_0.AdrDriveStatus := ADR (DriveStatus);
		MC_BR_ReadDriveStatus_0();
		gA[12].Ind_Simulation		:=	DriveStatus.Simulation;
		gA[12].Ind_NetworkInit		:=	DriveStatus.NetworkInit;
		gA[12].Input_Home			:=	DriveStatus.HomeSwitch;
		gA[12].Input_PosHW			:=	DriveStatus.PosHWSwitch;
		gA[12].Input_NegHW			:=	DriveStatus.NegHWSwitch;
		gA[12].Input_Trigger1		:=	DriveStatus.Trigger1;
		gA[12].Input_Trigger2		:=	DriveStatus.Trigger2;
		gA[12].Input_DriveEnable		:=	DriveStatus.DriveEnable;
		gA[12].Ind_ControllerReady	:=	DriveStatus.ControllerReady;
		gA[12].Ind_ControllerStatus	:=	DriveStatus.ControllerStatus;
		gA[12].Error					:=	DriveStatus.AxisError;
		gA[12].Ind_LagWarning		:=	DriveStatus.LagWarning;

	(************************ READ AXIS ERROR **********************)
		MC_ReadAxisError_0.Enable := gA[12].Ind_NetworkInit;
		MC_ReadAxisError_0.Axis := gA[12].Ident;
		MC_ReadAxisError_0.DataAddress := ADR(gA[12].ErrorText);
		MC_ReadAxisError_0.DataLength := SIZEOF(gA[12].ErrorText);
		MC_ReadAxisError_0.DataObjectName := 'Error_Eng';
		MC_ReadAxisError_0();
		IF(MC_ReadAxisError_0.Valid) THEN
			gA[12].ErrorID := MC_ReadAxisError_0.AxisErrorID;
			gA[12].ErrorCount := MC_ReadAxisError_0.AxisErrorCount;
		END_IF
	(* Auto Acknowledge Errors *)
		IF (gA[12].Cmd_Reset AND (gA[12].ErrorCount<>0) AND NOT AutoAck) THEN
			AutoAck:=1;
		ELSE
			AutoAck:=0;
		END_IF
	(*Axis Error Acknowledge*)
		IF (EDGEPOS(AutoAck) OR EDGEPOS(gA[12].ErrorAck)) THEN
			MC_ReadAxisError_0.Acknowledge := 1;
		ELSE;
			MC_ReadAxisError_0.Acknowledge :=0;
		END_IF

	(************************ RESET AXIS ERROR **********************)
		IF (gA[12].Cmd_Reset AND (gA[12].ErrorCount=0) AND gA[12].ErrorStop) THEN
			MC_Reset_0.Execute:=1;
		END_IF
		IF (MC_Reset_0.Done) THEN
			MC_Reset_0.Execute:=0;
			gA[12].Cmd_Reset:=0;
			ResetError := 0;
		END_IF
		IF (MC_Reset_0.Error) THEN
			MC_Reset_0.Execute:=0;
			gA[12].Cmd_Reset:=0;
			ResetError := 1;
		END_IF
		MC_Reset_0.Axis:=gA[12].Ident;
		MC_Reset_0();

	(************************ READ AXIS STATUS *************************)
		MC_ReadStatus_0.Enable := gA[12].Ind_NetworkInit;
		MC_ReadStatus_0.Axis := gA[12].Ident;
		MC_ReadStatus_0();
		IF(MC_ReadStatus_0.Valid = TRUE)THEN
			gA[12].Ind_Enabled 			     := NOT (MC_ReadStatus_0.Disabled);
			gA[12].Ind_StandStill		     := MC_ReadStatus_0.StandStill;
			gA[12].Ind_Stopping		    	 := MC_ReadStatus_0.Stopping;
			gA[12].Ind_DiscreteMotion	   := MC_ReadStatus_0.DiscreteMotion;
			gA[12].Ind_ContinuousMotion	 := MC_ReadStatus_0.ContinuousMotion;
			gA[12].Ind_SynchronizedMotion := MC_ReadStatus_0.SynchronizedMotion;
			gA[12].ErrorStop := MC_ReadStatus_0.Errorstop;
		END_IF
    IF NOT(gA[12].Ind_Enabled) THEN
      gA[12].bSynchroReq := 1 ;
    END_IF
    IF EDGEPOS(gA[12].Ind_bSynchroOK) THEN
      gA[12].bSynchroReq := 0 ;
    END_IF

	(******************** INIT POSITION MODULUS  *********************)
    IF ( gA[12].Ind_StandStill     OR
         NOT(gA[12].Ind_Enabled) ) AND
         g_bChangeModTearEBReq     THEN
      bChangeModReq := 1 ;
      uiInitModPos0_ErrorID := 0 ;
    END_IF
    MC_BR_InitModPos_0.Execute:= (InitModPosition OR bChangeModReq) ;
		MC_BR_InitModPos_0.Axis:= gA[12].Ident;
		MC_BR_InitModPos_0.Period:= REAL_TO_UDINT(gA[12].AxisPeriod);
		MC_BR_InitModPos_0.Factor:=1;
		InitModPos_Done:=MC_BR_InitModPos_0.Done;

    IF MC_BR_InitModPos_0.Done THEN
      g_bChangeModTearEBReq := 0 ;
      bChangeModReq         := 0 ;
    ELSIF MC_BR_InitModPos_0.Error THEN
      bChangeModReq := 0 ;
      uiInitModPos0_ErrorID := MC_BR_InitModPos_0.ErrorID ;
    END_IF
		MC_BR_InitModPos_0();

	(******************** INIT ENDLESS POSITION *********************)
		MC_BR_InitEndlessPosition_0.Execute:= InitModPos_Done;
		MC_BR_InitEndlessPosition_0.Axis:= gA[12].Ident;
		MC_BR_InitEndlessPosition_0.DataAddress:= ADR(gEndPosData[12]);
		IF (MC_BR_InitEndlessPosition_0.Done) THEN
			InitModPosition:=0;
			InitEndlessPosition:=0;
			HomeRestore:=1;
		END_IF
		MC_BR_InitEndlessPosition_0();

	(************************ HOME AXIS FIRST POWER UP **********************)
		IF (HomeRestore AND NOT gA12_FirstHomed) THEN
			MC_Home_0.Execute:=1;
		END_IF
		MC_Home_0.Axis:=gA[12].Ident;
		MC_Home_0.Position:=0;
		MC_Home_0.HomingMode:=mcHOME_DIRECT;
		IF (MC_Home_0.Done) THEN
			MC_Home_0.Execute:=0;
			gA12_FirstHomed:=1;
		END_IF
		MC_Home_0();

  (************************ HOME AXIS **********************)
    IF (gA12_FirstHomed) THEN
      MC_Home_1.Execute:=HomeRestore;
    END_IF
    MC_Home_1.Axis:=gA[12].Ident;
    MC_Home_1.Position:=0;
    MC_Home_1.HomingMode:=mcHOME_RESTORE_POS;
    IF (MC_Home_1.Done) THEN
      gA[12].Ind_Homed:=1;
      HomeRestore:=0;
    END_IF
    MC_Home_1();

	(******************** READ ACTUAL POSITION *********************)
		MC_ReadActualPosition_0.Enable:= gA[12].Ind_NetworkInit;
		MC_ReadActualPosition_0.Axis:= gA[12].Ident;
		MC_ReadActualPosition_0();
		IF(MC_ReadActualPosition_0.Valid = TRUE)THEN
			gA[12].PositionCount := MC_ReadActualPosition_0.Position;
			gA[12].PositionInch := gA[12].PositionCount/gA[12].UnitsPerInch;
			gA[12].PositionDeg := gA[12].PositionCount/gA[12].UnitsPerDeg;
		END_IF

  //******************** READ SET POINT POSITION *********************
    // Slave side  : ParID 428 SGEN_S_SET : CTRL Position controller: Input set position
    // Master side : ParID 412 S_SET_VAX1 : 412: VAX: Position

    // Slave side
    MC_BR_CyclicRead_0.Axis        := gA[12].Ident ;
    MC_BR_CyclicRead_0.Enable      := gA[12].Ind_NetworkInit;
    MC_BR_CyclicRead_0.ParID       := 428 ;
    MC_BR_CyclicRead_0.DataAddress := ADR(iiSP_SlPos_U);
    MC_BR_CyclicRead_0.DataType    := ncPAR_TYP_DINT ;
    // Master side
    MC_BR_CyclicRead_1.Axis        := gA[9].Ident ;
    MC_BR_CyclicRead_1.Enable      := gA[12].Ind_NetworkInit;
    MC_BR_CyclicRead_1.ParID       := 412 ;
    MC_BR_CyclicRead_1.DataAddress := ADR(iiSP_MaPos_U);
    MC_BR_CyclicRead_1.DataType    := ncPAR_TYP_DINT ;

    IF MC_BR_CyclicRead_0.Valid THEN
      rSP_SlPos_Deg := iiSP_SlPos_U/gA[12].UnitsPerDeg ;
    ELSIF MC_BR_CyclicRead_0.Error THEN
      MC_BR_CyclicRead_0.Enable := 0 ;
    END_IF
    IF MC_BR_CyclicRead_1.Valid THEN
      rSP_MaPos_Deg := iiSP_MaPos_U/gA[9].UnitsPerDeg ;
    ELSIF MC_BR_CyclicRead_1.Error THEN
      MC_BR_CyclicRead_1.Enable := 0 ;
    END_IF
    MC_BR_CyclicRead_0();
    MC_BR_CyclicRead_1();

  //******************** READ ACTUAL SLAVE PHASE *********************
  IF gA[12].rRSynDen > 0.0 THEN
    rTempActPhasDeg := rSP_SlPos_Deg
                       - gA[12].rRSynNum / gA[12].rRSynDen
                       * rSP_MaPos_Deg;
    gA[12].rActPhasDeg := H_FC_Modulus (
                              IN_rMod := 360 * gA[12].rRSynNum / gA[12].rRSynDen ,
                              IN_rVar := rTempActPhasDeg
                                      ) ;
  END_IF

	(******************** READ ACTUAL VELOCITY *********************)
		IF(MC_ReadActualVelocity_0.Error=TRUE) THEN
			MC_ReadActualVelocity_0.Enable:= 0;
		ELSE
			MC_ReadActualVelocity_0.Enable:= 1;
		END_IF
		MC_ReadActualVelocity_0.Axis:= gA[12].Ident;
		MC_ReadActualVelocity_0();
		IF(MC_ReadActualVelocity_0.Valid = TRUE)THEN
      //gA[12].ActualVelocity := MC_ReadActualVelocity_0.Velocity*60/gA[12].SP_MotorPPR;
      gA[12].ActualVelocity := MC_ReadActualVelocity_0.Velocity*60/gA[12].AxisPeriod ; // D.M. 03/08/2011 BrownPaper_14542  Need speed of the axis and not of the shaft of the motor
			IF ABS(gA[12].ActualVelocity>1) THEN // D.M. 03/08/2011 BrownPaper_14542 Add ABS because in case negative velocity Ind_InMotion = 0 instead of 1
				gA[12].Ind_InMotion:=1;
			ELSE
				gA[12].Ind_InMotion:=0;
			END_IF
		END_IF

	(******************** READ ACTUAL TORQUE *********************)
		IF(MC_ReadActualTorque_0.Error=TRUE) THEN
			MC_ReadActualTorque_0.Enable:= 0;
		ELSE
			MC_ReadActualTorque_0.Enable:= 1;
		END_IF
		MC_ReadActualTorque_0.Axis:= gA[12].Ident;
		MC_ReadActualTorque_0();
		IF(MC_ReadActualTorque_0.Valid = TRUE)THEN
			gA[12].ActualTorque := MC_ReadActualTorque_0.Torque;
		END_IF

	(************************ ENABLE AXIS **********************)
		MC_Power_0.Axis:=gA[12].Ident;
		IF (MC_Power_0.Error=0) THEN
			MC_Power_0.Enable:=gA[12].Cmd_Enable;
		ELSE;
			MC_Power_0.Enable:=0;
		END_IF;
		MC_Power_0();

	(************************ AXIS VELOCITY MOVE **********************)
		MC_MoveVelocity_0.Axis:=gA[12].Ident;
		MC_MoveVelocity_0.Velocity:=gA[12].SP_Velocity*gA[12].AxisPeriod/60;
		MC_MoveVelocity_0.Acceleration:=gA[12].SP_Accel;
		MC_MoveVelocity_0.Deceleration:=gA[12].SP_Decel;
		MC_MoveVelocity_0.Direction:=mcPOSITIVE_DIR;
		IF ((EDGEPOS(gA[12].Cmd_ContinuousMotion)) OR (EDGEPOS(gA[12].Cmd_ContinuousMotionUpdate))) THEN
			MC_MoveVelocity_0.Execute:=1;
		ELSE
			MC_MoveVelocity_0.Execute:=0;
		END_IF;
		MC_MoveVelocity_0();

  //************************ AXIS OVERRIDE **********************
    MC_SetOverride_0.Axis      := gA[12].Ident ;
    MC_SetOverride_0.Enable    := gA[12].Cmd_Override ;
    MC_SetOverride_0.VelFactor := gA[12].rSP_OverrideV ;
    MC_SetOverride_0.AccFactor := gA[12].rSP_OverrideA ;
    IF (MC_SetOverride_0.Enabled) OR
       (MC_SetOverride_0.Error)   THEN
      gA[12].Cmd_Override := 0 ;
    END_IF
    MC_SetOverride_0();

  (************************ AXIS HALT **********************)
    MC_Halt_0.Axis:=gA[12].Ident;
    MC_Halt_0.Deceleration := gA[12].SP_Decel ;
    MC_Halt_0.Execute      := gA[12].Cmd_Halt;
    IF (MC_Halt_0.Done OR MC_Halt_0.CommandAborted OR MC_Halt_0.Error) THEN
      MC_Halt_0.Execute:=0;
      uiMC_Halt_0_MemoErrorID := MC_Halt_0.ErrorID ;
    END_IF;
    MC_Halt_0();

  (************************ AXIS STOP **********************)
    MC_Stop_0.Axis:=gA[12].Ident;
    IF (gA[12].Ind_ContinuousMotion AND (NOT gA[12].Cmd_ContinuousMotion) AND gAlarmsOK) THEN
      MC_Stop_0.Deceleration:=gA[12].SP_Decel;
      MC_Stop_0.Execute:=1;
    END_IF;
    IF (MC_Stop_0.Done OR MC_Stop_0.CommandAborted OR MC_Stop_0.Error) THEN
      MC_Stop_0.Execute:=0;
    END_IF;
    MC_Stop_0();

  (************************  ESTOP **********************)
    MC_Stop_1.Axis:=gA[12].Ident;
    IF EDGEPOS(g_bIndEStopStandstill) THEN
      MC_Stop_1.Deceleration:=gA[12].SP_EStopDecel;
      MC_Stop_1.Execute:=1;
    END_IF;
    IF (MC_Stop_1.Done OR MC_Stop_1.CommandAborted OR MC_Stop_1.Error) THEN
      MC_Stop_1.Execute:=0;
      gA[12].Cmd_EStopDisable := 1 ;
    END_IF;
    IF NOT(g_bIndEStopStandstill) THEN
      gA[12].Cmd_EStopDisable := 0 ;
    END_IF;
    MC_Stop_1();

    (************************ AXIS PHASE CONTROL (Inches) First Step **********************)
    IF EDGEPOS(gA[12].Cmd_PhaseOffset) THEN
      rSP_PhaseOffset := gA[12].SP_PhaseOffset ;
    END_IF;

    (************************ SHIFTING PERF CONTROL **********************)
    IF g_bCmdShiftA[12] THEN
      //rSP_ShiftEnvB := g_iPerfShiftPos * gr_rIncrShiftPerf_mm/25.4 * gA[12].rRSynNum/gA[12].rRSynDen ; // D.M. RS26_Pyrollpack_14661 CAUTION !!! Phasing acts on the master side and not slave side, replaced by the code below
      rSP_ShiftEnvB := g_iPerfShiftPos * gr_rIncrShiftPerf_mm/25.4 ;
      gA[12].Cmd_PhaseOffset := 1 ;
      g_bCmdShiftA[12] := 0 ;
    END_IF

    (************************ AXIS PHASE CONTROL (Inches) Next Step **********************)
    MC_BR_Phasing_0.Slave:=gA[12].Ident;
    IF gA[12].Ind_SynchronizedMotion AND NOT(gstCycA[12].CycManTimSet.bSCyc) AND st_TON_0.Q THEN
      MC_BR_Phasing_0.Enable:=1;
    ELSE
      MC_BR_Phasing_0.Enable:=0;
    END_IF
    IF gA[12].Cmd_PhaseOffset              AND
       EDGENEG(gA[12].Ind_bInContactZone)  AND
       NOT(gstCycA[12].CycManTimSet.bSCyc) THEN
      MC_BR_Phasing_0.InitData := 1 ;
      gA[12].Cmd_PhaseOffset := 0 ;
      rSP_PhaseOffsetVal := rSP_PhaseOffset + rSP_ShiftEnvB ;
      // Calculation new phase Holding/Master
      rTemp_[0] := (rSP_PhaseOffsetVal)/gA[12].InchPerDeg ;
      rTemp_[1] := gRecipeActive.rEnvB_PhasMasterDeg + rTemp_[0]*gA[12].rRSynNum/gA[12].rRSynDen ;
      gRecipeActive.rEnvB_PhasMasterDeg := H_FC_Modulus (IN_rMod := 360*gA[12].rRSynNum/gA[12].rRSynDen, IN_rVar := rTemp_[1]) ;
      rSP_ShiftEnvB := 0.0 ;
      rSP_PhaseOffset := 0.0 ;
      iTest_[0] := iTest_[0] + 1 ;
      rTest_[iTest_[0]] := rTemp_[0] ;
    ELSE
      MC_BR_Phasing_0.InitData:=0;
    END_IF
    MC_BR_Phasing_0.Shift               := rSP_PhaseOffsetVal*gA[9].UnitsPerInch;
    MC_BR_Phasing_0.Velocity            := 6*gA[12].AxisPeriod/60;
    MC_BR_Phasing_0.Acceleration        := gA[12].SP_Decel;
    MC_BR_Phasing_0.ApplicationDistance := 0.8*gA[9].AxisPeriod * gA[12].rRSynNum/gA[12].rRSynDen;
    MC_BR_Phasing_0.ApplicationMode     := mcMASTER_DISTANCE_BASED;
    MC_BR_Phasing_0.ShiftMode           := mcRELATIVE;
    MC_BR_Phasing_0();

    (************************ AXIS PHASE CONTROL (Inches) TIMING SETTING **********************)
    IF gstCycA[12].CycManTimSet.bSCyc THEN
      IF gA[12].Cmd_ManuTimSetPlus THEN
        rAxisTimSet_SP_Vel := gr_rAxisTimSet_SP_Vel*gA[9].AxisPeriod/60 / (gA[12].rRSynNum/gA[12].rRSynDen) ;
      ELSE
        rAxisTimSet_SP_Vel := - gr_rAxisTimSet_SP_Vel*gA[9].AxisPeriod/60 / (gA[12].rRSynNum/gA[12].rRSynDen) ;
      END_IF
        rAxisTimSet_SP_Acc := gr_rAxisTimSet_SP_Acc*gA[9].AxisPeriod/60/60 / (gA[12].rRSynNum/gA[12].rRSynDen) ;
    END_IF

    MC_BR_Phasing_1.Slave                  := gA[12].Ident;
    MC_BR_Phasing_1.Enable                 := gstCycA[12].CycManTimSet.bCyc ;
    MC_BR_Phasing_1.InitData               := gstCycA[12].CycManTimSet.bSCyc ;
    MC_BR_Phasing_1.PerformVelocityControl := gstCycA[12].CycManTimSet.CmdMov ;
    MC_BR_Phasing_1.Velocity               := rAxisTimSet_SP_Vel ;
    MC_BR_Phasing_1.Acceleration           := rAxisTimSet_SP_Acc ;
    MC_BR_Phasing_1.ApplicationMode        := mcVELOCITY_CONTROL ;
    MC_BR_Phasing_1();
    st_TON_0(IN:=NOT(MC_BR_Phasing_1.Enable),PT:=T#100ms) ;

    IF NOT(gstCycA[12].CycManTimSet.CmdMov) AND
       MC_BR_Phasing_1.ShiftAttained       OR
       NOT(gstCycA[12].CycManTimSet.bCyc)   OR
       MC_BR_Phasing_1.Error               AND
       1                                   THEN
      gstCycA[12].CycManTimSet.CmdStop := 0 ;
    END_IF
	END_IF

END_PROGRAM
```

#### A12_BasicInit.st - Initialization code
```iecst
(********************************************************************
 * COPYRIGHT -- Microsoft
 ********************************************************************
 * Program: A12_Basic
 * File: A12_BasicInit.st
 * Author: dominique
 * Created: November 21, 2011
 ********************************************************************
 * Implementation of program A12_Basic
 ********************************************************************)

PROGRAM _INIT

	(* Axis Setpoint Variables *)
		gA[12].SP_MotorPPR := 36000 / 6 ; // One revolution on the shaft = 1/2 revolution of the Axis. When Axis perfoms 1 rev shaft performs 2 rev. One Axis rev = 2 shaft rev = 1 bag
		gA[12].SP_GearBoxInput:= 6;
		gA[12].SP_GearBoxOutput:= 1;
		gA[12].AxisPeriod := gA[12].SP_MotorPPR*gA[12].SP_GearBoxInput/gA[12].SP_GearBoxOutput ;
		gA[12].UnitsPerDeg := gA[12].AxisPeriod/360;
		gA[12].SP_Accel := 0.2*gA[12].AxisPeriod;
		gA[12].SP_Decel := 0.4*gA[12].AxisPeriod;
		gA[12].SP_EStopDecel := 1000.0*gA[12].AxisPeriod; // Stop axis from 1000 tr/min in 1s
		gA[12].HomeVelocity := 6*gA[12].AxisPeriod/60;
    gA[12].rSP_CorPosVel := 0.0 ;
    gA[12].rSP_OverrideV := 1.0 ;
    gA[12].rSP_OverrideA := 1.0 ;
    gA[12].Cmd_EStopDisable := 0 ;

	(* access master axis *)
		AxisErrorNcAccess := ncaccess(ncACP10MAN, ADR('Axis12'), ADR(gA[12].Ident));

	(* Trigger Initialization Of ModPosition *)
		InitModPosition:=1;

END_PROGRAM
```

#### A12_Basic.var - Local variables
```iecst
(********************************************************************
 * COPYRIGHT -- Microsoft
 ********************************************************************
 * Program: A12_Basic
 * File: A12_Basic.var
 * Author: dominique
 * Created: November 21, 2011
 ********************************************************************
 * Local variables of program A12_Basic
 ********************************************************************)
VAR
	AutoAck : BOOL;
	AxisErrorNcAccess : UINT;
	DriveStatus : MC_DRIVESTATUS_TYP;
	HomeRestore : BOOL;
	InitEndlessPosition : BOOL;
	InitModPos_Done : BOOL;
	InitModPosition : BOOL;
	MC_BR_InitEndlessPosition_0 : MC_BR_InitEndlessPosition;
	MC_BR_InitModPos_0 : MC_BR_InitModPos;
  uiInitModPos0_ErrorID : UINT ;
  MC_BR_Phasing_0 : MC_BR_Phasing;
  MC_BR_Phasing_1 : MC_BR_Phasing;
	MC_BR_ReadDriveStatus_0 : MC_BR_ReadDriveStatus;
	MC_Home_0 : MC_Home;
  MC_Home_1 : MC_Home;
  MC_Home_2 : MC_Home;
	MC_MoveVelocity_0 : MC_MoveVelocity;
	MC_Power_0 : MC_Power;
	MC_ReadActualPosition_0 : MC_ReadActualPosition;
	MC_ReadActualTorque_0 : MC_ReadActualTorque;
	MC_ReadActualVelocity_0 : MC_ReadActualVelocity;
	MC_ReadAxisError_0 : MC_ReadAxisError;
	MC_ReadStatus_0 : MC_ReadStatus;
	MC_Reset_0 : MC_Reset;
  MC_Halt_0 : MC_Halt ;
  uiMC_Halt_0_MemoErrorID : UINT ;
  MC_Stop_0 : MC_Stop;
  MC_Stop_1 : MC_Stop;
  st_TON_0 : TON ;
	ResetError : BOOL;
  rAxisTimSet_SP_Vel  : REAL ; (*Set point Velocity for Axis manual timing setting cycle, in units/s*)
  rAxisTimSet_SP_Acc  : REAL ; (*Set point Acceleration for Axis manual timing setting cycle, in units/s²*)
  rAxisTimSet_SP_Dec  : REAL ; (*Set point Deceleration for Axis manual timing setting cycle, in units/s²*)
  uiAxisTimSet_SP_Dir : USINT ; (*Set point Direction for Axis manual timing setting cycle*)
  uiAxisTimSet_SP_ShiftAppMode : UINT ; (*Set point Shit Application mode for phasing Axis manual timing setting cycle*)
  rTempActPhasDeg : REAL;
  iTest_ : ARRAY[0..9] OF INT ;
  rTest_ : ARRAY[0..9] OF REAL ;
  rTemp_ : ARRAY[0..9] OF REAL ;
  rA9PosCorDeg  : REAL;
  rRepeatMetric : REAL;
  MC_SetOverride_0 : MC_SetOverride;

  iiSP_SlPos_U  : DINT ; (*On Slave side, input set point position of the position controller ParID 428, in unit*)
  rSP_SlPos_Deg : REAL ; (*On Slave side, input set point position of the position controller ParID 428, in deg*)
  iiSP_MaPos_U  : DINT ; (*On Master side, input set point position of the position controller ParID 412, in unit*)
  rSP_MaPos_Deg : REAL ; (*On Master side, input set point position of the position controller ParID 412, in deg*)
  MC_BR_CyclicRead_0 : MC_BR_CyclicRead ;
  MC_BR_CyclicRead_1 : MC_BR_CyclicRead ;

  bChangeModReq      : BOOL ;
  rRedefPosTear      : REAL ;
  rPosTear4Pliers    : REAL ;
  rSP_PhaseOffset    : REAL ;
  rSP_PhaseOffsetVal : REAL ;
  rSP_ShiftEnvB      : REAL ;

  rA12PosTempAxis_deg : REAL;
END_VAR
```

### Program Logical/BagMachine_Section/EnvBag/Axis12/A12_Control (IEC) - Servo Control

#### A12_Control.var
```iecst
(********************************************************************
 * COPYRIGHT -- Microsoft
 ********************************************************************
 * Program: A12_Control
 * File: A12_Control.var
 * Author: dominique
 * Created: November 21, 2011
 ********************************************************************
 * Local variables of program A12_Control
 ********************************************************************)
VAR
	HGW_ChangeReal_0 : HGW_ChangeReal;
	HGW_RelativeChangeReal1_0 : H_FB_RelativeChangeLimitReal1;
	HGW_Toggle_0 : HGW_Toggle;
	Synch_Permissive : BOOL;
	TOF_0 : TOF;
	TON_0 : TON;
  rIncrOffsetAxeRun_Inch : REAL ;
END_VAR
```

### Program Logical/BagMachine_Section/EnvBag/Axis12/A12_Ref (IEC) - Reference Routine

#### A12_RefCyclic.ld
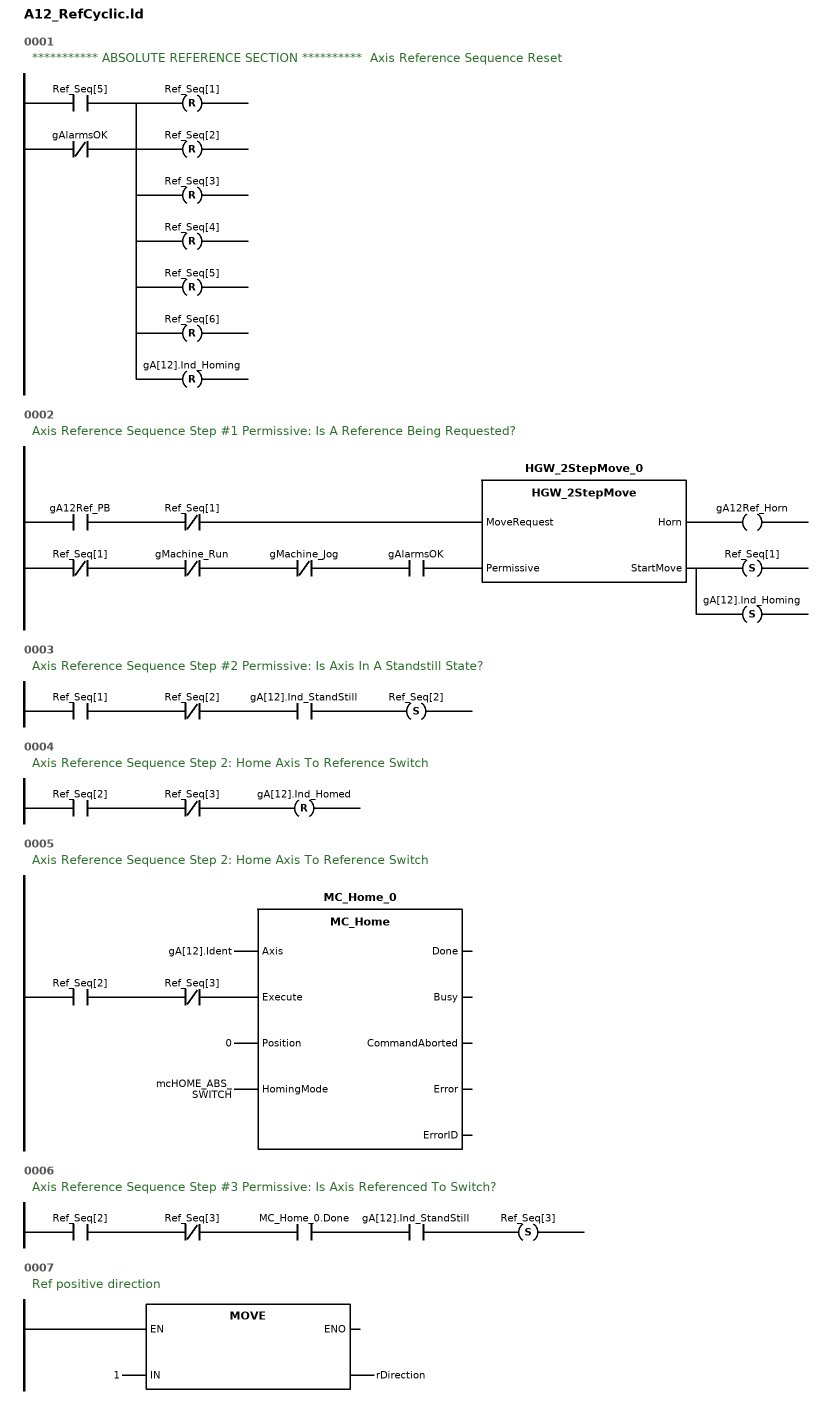
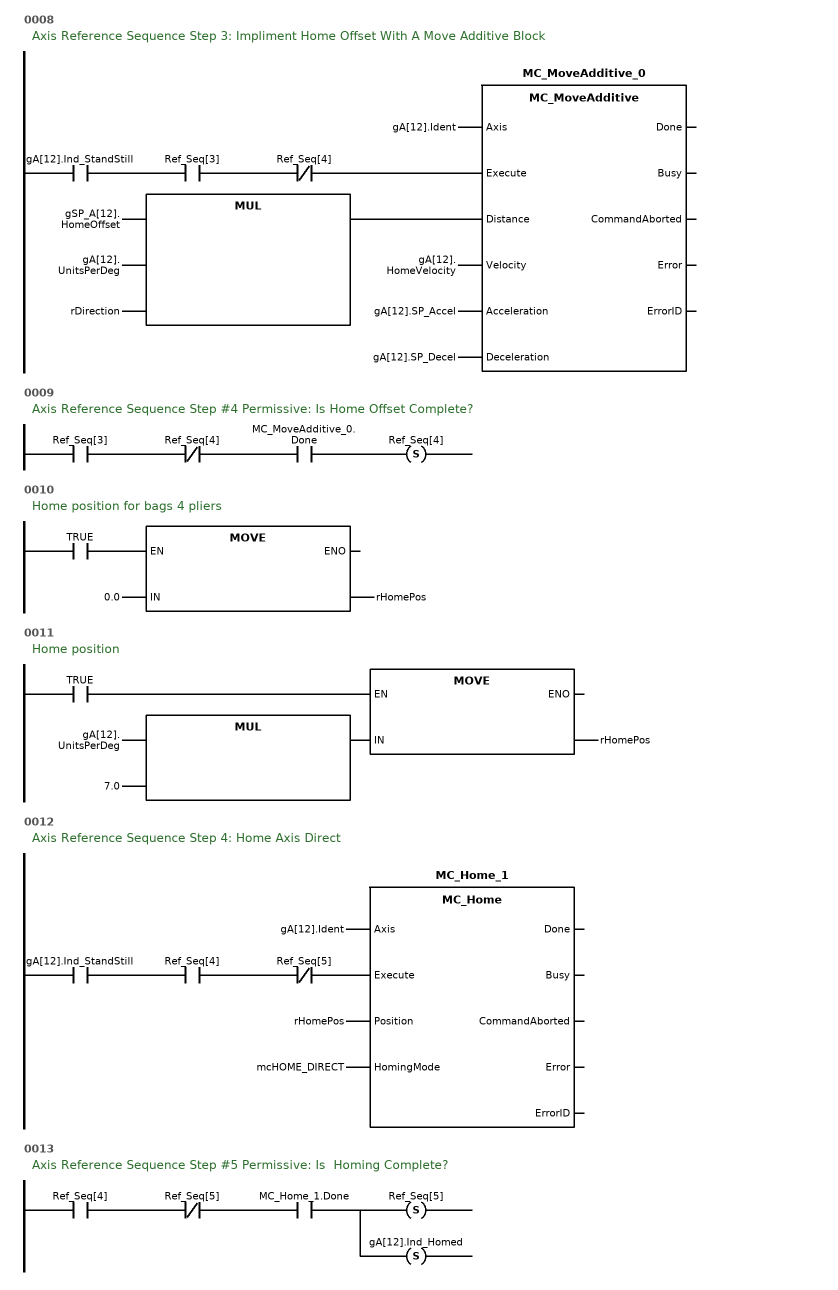
Ladder, written as Structured Text:
```iecst
(********************************************************************
 * COPYRIGHT -- Microsoft
 ********************************************************************
 * Program: A4_Ref
 * File: A4_RefCyclic.ld
 * Author: pkiel
 * Created: July 19, 2011
 ********************************************************************
 * Implementation of program A4_Ref
 ********************************************************************)

PROGRAM _CYCLIC
VAR
    _p1 : BOOL;
    _p2 : BOOL;
END_VAR
(* Network 1: *********** ABSOLUTE REFERENCE SECTION **********  Axis Reference Sequence Reset *)
_p1 := Ref_Seq[5];
IF Ref_Seq[5] OR NOT gAlarmsOK THEN Ref_Seq[1] := FALSE; END_IF;
IF _p1 OR NOT gAlarmsOK THEN
    Ref_Seq[2] := FALSE;
    Ref_Seq[3] := FALSE;
    Ref_Seq[4] := FALSE;
    Ref_Seq[5] := FALSE;
    Ref_Seq[6] := FALSE;
    gA[12].Ind_Homing := FALSE;
END_IF;

(* Network 2: Axis Reference Sequence Step #1 Permissive: Is A Reference Being Requested? *)
HGW_2StepMove_0(MoveRequest := gA12Ref_PB AND NOT Ref_Seq[1], Permissive := NOT Ref_Seq[1] AND NOT gMachine_Run AND NOT gMachine_Jog AND gAlarmsOK);
gA12Ref_Horn := HGW_2StepMove_0.Horn;
IF HGW_2StepMove_0.StartMove THEN
    Ref_Seq[1] := TRUE;
    gA[12].Ind_Homing := TRUE;
END_IF;

(* Network 3: Axis Reference Sequence Step #2 Permissive: Is Axis In A Standstill State? *)
IF Ref_Seq[1] AND NOT Ref_Seq[2] AND gA[12].Ind_StandStill THEN Ref_Seq[2] := TRUE; END_IF;

(* Network 4: Axis Reference Sequence Step 2: Home Axis To Reference Switch *)
IF Ref_Seq[2] AND NOT Ref_Seq[3] THEN gA[12].Ind_Homed := FALSE; END_IF;

(* Network 5: Axis Reference Sequence Step 2: Home Axis To Reference Switch *)
MC_Home_0(Axis := gA[12].Ident, Execute := Ref_Seq[2] AND NOT Ref_Seq[3], Position := 0, HomingMode := mcHOME_ABS_SWITCH);

(* Network 6: Axis Reference Sequence Step #3 Permissive: Is Axis Referenced To Switch? *)
IF Ref_Seq[2] AND NOT Ref_Seq[3] AND MC_Home_0.Done AND gA[12].Ind_StandStill THEN
    Ref_Seq[3] := TRUE;
END_IF;

(* Network 7: Ref positive direction  *)
rDirection := 1;

(* Network 8: Axis Reference Sequence Step 3: Impliment Home Offset With A Move Additive Block *)
MC_MoveAdditive_0(Axis := gA[12].Ident, Execute := gA[12].Ind_StandStill AND Ref_Seq[3] AND NOT Ref_Seq[4], Distance := gSP_A[12].HomeOffset * gA[12].UnitsPerDeg * rDirection, Velocity := gA[12].HomeVelocity, Acceleration := gA[12].SP_Accel, Deceleration := gA[12].SP_Decel);

(* Network 9: Axis Reference Sequence Step #4 Permissive: Is Home Offset Complete? *)
IF Ref_Seq[3] AND NOT Ref_Seq[4] AND MC_MoveAdditive_0.Done THEN Ref_Seq[4] := TRUE; END_IF;

(* Network 10: Home position for bags 4 pliers  *)
rHomePos := 0.0;

(* Network 11: Home position  *)
rHomePos := gA[12].UnitsPerDeg * 7.0;

(* Network 12: Axis Reference Sequence Step 4: Home Axis Direct *)
MC_Home_1(Axis := gA[12].Ident, Execute := gA[12].Ind_StandStill AND Ref_Seq[4] AND NOT Ref_Seq[5], Position := rHomePos, HomingMode := mcHOME_DIRECT);

(* Network 13: Axis Reference Sequence Step #5 Permissive: Is  Homing Complete? *)
_p2 := Ref_Seq[4] AND NOT Ref_Seq[5] AND MC_Home_1.Done;
IF Ref_Seq[4] AND NOT Ref_Seq[5] AND MC_Home_1.Done THEN Ref_Seq[5] := TRUE; END_IF;
IF _p2 THEN gA[12].Ind_Homed := TRUE; END_IF;
END_PROGRAM
```
